// ---- POUs/BaseModule/ActionModule/motorModule/visu/motionModuleP1.TcVIS
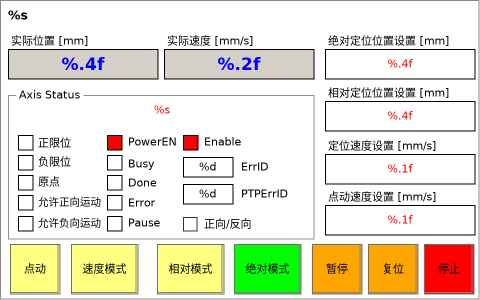
VISUALIZATION motionModuleP1  // 480x300
VAR_IN_OUT
	userData: motionModuleDataHMI;	
END_VAR
    Button (10,244 50x50), "点动", input disabled if: NOT userData.jogCondition OR NOT userData.ctrlModeCondition
        tap userData.manJogGo
    Button (157,244 67x50), "相对模式", tooltip "Please keep pressing to trigger", input disabled if: NOT userData.relCondition OR NOT userData.ctrlModeCondition
        tap userData.manRelGo
    Button (234,244 67x50), "绝对模式", tooltip "Please keep pressing to trigger", input disabled if: NOT userData.absCondition OR NOT userData.ctrlModeCondition
        tap userData.manABSGo
    Button (424,244 50x50), "停止"
        tap userData.stop
    Rectangle (8,49 150x30), "%.4f", text variable: userData.actualPos
    Rectangle (8,26 150x30), "实际位置 [mm]"
    Rectangle (164,49 150x30), "%.2f", text variable: userData.actualVel
    Rectangle (164,26 150x30), "实际速度 [mm/s]"
    Rectangle (325,79 145x28), "相对定位位置设置 [mm]"
    Rectangle (325,26 150x30), "绝对定位位置设置 [mm]"
    Rectangle (325,131 150x30), "定位速度设置 [mm/s]"
    GroupBox (8,87 306x152), "Axis Status"
        Rectangle (99,48 15x15), colour toggle: userData.powerEnable
        Rectangle (117,44 64x22), "PowerEN"
        Rectangle (10,48 15x15), colour toggle: userData.forwardLimitSwitch
        Rectangle (10,68 15x15), colour toggle: userData.backwardsLimitSwitch
        Rectangle (10,88 15x15), colour toggle: userData.dogPointSwitch
        Rectangle (27,84 64x22), "原点"
        Rectangle (99,68 15x15), colour toggle: userData.busy
        Rectangle (117,66 64x22), "Busy"
        Rectangle (230,69 46x22), "ErrID"
        Rectangle (27,104 67x22), "允许正向运动"
        Rectangle (10,108 15x15), colour toggle: userData.forwardEnable
        Rectangle (27,125 67x22), "允许负向运动"
        Rectangle (10,129 15x15), colour toggle: userData.backwardsEnable
        Rectangle (117,85 64x22), "Done"
        Rectangle (117,105 64x22), "Error"
        Rectangle (175,97 50x20), "%d", text variable: userData.PTPErrID
        Rectangle (99,129 15x15), colour toggle: userData.oPause
        Rectangle (117,125 64x22), "Pause"
        Rectangle (27,45 68x22), "正限位"
        Rectangle (27,64 64x22), "负限位"
        Rectangle (175,70 50x20), "%d", text variable: userData.errID
        Rectangle (175,48 15x15), colour toggle: userData.enable
        Rectangle (230,96 64x22), "PTPErrID"
        Rectangle (99,88 15x15), colour toggle: userData.done
        Rectangle (99,108 15x15), colour toggle: userData.error
        Checkbox (173,122 130x30), "正向/反向", variable: userData.choiceOfDirection
        Rectangle (193,44 52x22), "Enable"
    Rectangle (12,100 300x20), "%s", text variable: userData.errTxt
    Rectangle (325,49 150x30), "%.4f", text variable: userData.manABSPos, input disabled if: Not userData.goHomeDone
        OnMouseDown: write the text variable via Edit
    Rectangle (325,101 150x30), "%.4f", text variable: userData.manRelDis
        OnMouseDown: write the text variable via Edit
    Rectangle (325,154 150x30), "%.1f", text variable: userData.manVel
        OnMouseDown: write the text variable via Edit
    Rectangle (325,182 150x30), "点动速度设置 [mm/s]"
    Rectangle (325,205 150x30), "%.1f", text variable: userData.manJogVel
        OnMouseDown: write the text variable via Edit
    Button (71,244 67x50), "速度模式", invisible if: FALSE, input disabled if: NOT userData.velCondition OR NOT userData.ctrlModeCondition
        tap userData.manVelGo
    Button (368,244 50x50), "复位"
        tap userData.reset
    Rectangle (5,5 467x20), "%s", text variable: userData.nameTXT
    Button (312,244 50x50), "暂停", colour toggle: userData.oPause, input disabled if: NOT userData.ctrlModeCondition
        tap userData.pauseB
END_VISUALIZATION

// ---- POUs/BaseModule/ActionModule/motorModule/visu/motionModuleP2.TcVIS
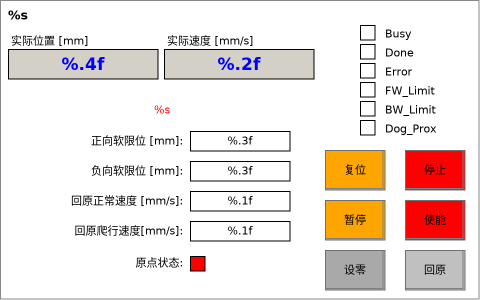
VISUALIZATION motionModuleP2  // 480x300
VAR_IN_OUT
	userData: motionModuleDataHMI;
END_VAR
    Rectangle (36,126 150x30), "正向软限位 [mm]:"
    Rectangle (190,131 100x20), "%.3f", text variable: userData.softPLimitPos, input disabled if: TRUE
        OnMouseDown: write the text variable via Edit
    Rectangle (36,156 150x30), "负向软限位 [mm]:"
    Rectangle (190,161 100x20), "%.3f", text variable: userData.softNLimitPos, input disabled if: TRUE
        OnMouseDown: write the text variable via Edit
    Rectangle (190,191 100x20), "%.1f", text variable: userData.goHomeVel
        OnMouseDown: write the text variable via Edit
    Button (405,250 60x40), "回原", colour toggle: userData.goHomeDone, input disabled if: NOT userData.homeCondition OR NOT userData.ctrlModeCondition
        tap userData.goHomeGo
    Rectangle (190,221 100x20), "%.1f", text variable: userData.goHomeVelSlow
        OnMouseDown: write the text variable via Edit
    Rectangle (36,186 150x30), "回原正常速度 [mm/s]:"
    Rectangle (27,216 159x30), "回原爬行速度[mm/s]:"
    Rectangle (79,248 107x30), "原点状态:"
    Rectangle (8,49 150x30), "%.4f", text variable: userData.actualPos
    Rectangle (8,26 150x30), "实际位置 [mm]"
    Rectangle (164,49 150x30), "%.2f", text variable: userData.actualVel
    Rectangle (164,26 150x30), "实际速度 [mm/s]"
    Rectangle (360,82 15x15), colour toggle: userData.forwardLimitSwitch
    Rectangle (360,101 15x15), colour toggle: userData.backwardsLimitSwitch
    Rectangle (360,120 15x15), colour toggle: userData.dogPointSwitch
    Rectangle (382,80 64x22), "FW_Limit"
    Rectangle (382,99 64x22), "BW_Limit"
    Rectangle (382,118 64x22), "Dog_Prox"
    Button (405,200 60x40), "使能", colour toggle: userData.powerEnable, input disabled if: NOT userData.ctrlModeCondition
        tap userData.power
    Button (325,250 60x40), "设零", invisible if: TRUE, input disabled if: NOT userData.setCondition OR NOT userData.ctrlModeCondition
        tap userData.setZero
    Button (325,200 60x40), "暂停", colour toggle: userData.oPause, input disabled if: NOT userData.ctrlModeCondition
        tap userData.pauseB
    Rectangle (190,256 15x15), colour toggle: userData.goHomeDone
    Rectangle (12,100 300x20), "%s", text variable: userData.errTxt
    Rectangle (5,5 467x20), "%s", text variable: userData.nameTXT
    Button (405,150 60x40), "停止"
        tap userData.stop
    Button (325,150 60x40), "复位"
        tap userData.reset
    Rectangle (360,25 15x15), colour toggle: userData.busy
    Rectangle (382,23 64x22), "Busy"
    Rectangle (382,42 64x22), "Done"
    Rectangle (382,61 64x22), "Error"
    Rectangle (360,44 15x15), colour toggle: userData.done
    Rectangle (360,63 15x15), colour toggle: userData.error
END_VISUALIZATION

// ---- POUs/BaseModule/ActionModule/motorModule/visu/motionModuleP3.TcVIS
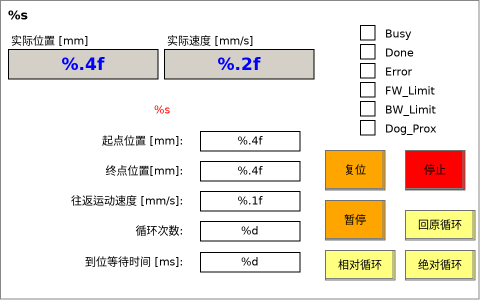
VISUALIZATION motionModuleP3  // 480x300
VAR_IN_OUT
	userData: motionModuleDataHMI;	
END_VAR
    Rectangle (36,126 150x30), "起点位置 [mm]:"
    Rectangle (36,156 150x30), "终点位置[mm]:"
    Rectangle (36,186 150x30), "往返运动速度 [mm/s]:"
    Rectangle (27,216 159x30), "循环次数:"
    Rectangle (8,49 150x30), "%.4f", text variable: userData.actualPos
    Rectangle (8,26 150x30), "实际位置 [mm]"
    Rectangle (164,49 150x30), "%.2f", text variable: userData.actualVel
    Rectangle (164,26 150x30), "实际速度 [mm/s]"
    Rectangle (12,100 300x20), "%s", text variable: userData.errTxt
    Rectangle (5,5 467x20), "%s", text variable: userData.nameTXT
    Rectangle (200,131 100x20), "%.4f", text variable: userData.loopFirstPoint
        OnMouseDown: write the text variable via Edit
    Rectangle (200,161 100x20), "%.4f", text variable: userData.loopSecondPoint
        OnMouseDown: write the text variable via Edit
    Rectangle (200,191 100x20), "%.1f", text variable: userData.loopGoVel
        OnMouseDown: write the text variable via Edit, min 0
    Rectangle (200,221 100x20), "%d", text variable: userData.loopCycle
        OnMouseDown: write the text variable via Edit, min 0
    Button (325,250 70x30), "相对循环", tooltip "Please keep pressing to trigger the relative motion loop", input disabled if: NOT userData.loopRelCondition OR NOT userData.ctrlModeCondition
        tap userData.loopRelGo
    Button (405,250 70x30), "绝对循环", tooltip "Please keep pressing to trigger the absolute motion loop", input disabled if: NOT userData.loopAbsCondition OR NOT userData.ctrlModeCondition
        tap userData.loopAbsGo
    Rectangle (27,247 159x30), "到位等待时间 [ms]:"
    Rectangle (200,252 100x20), "%d", text variable: userData.loopWatingTime
        OnMouseDown: write the text variable via Edit, min 0
    Button (405,150 60x40), "停止"
        tap userData.stop
    Button (325,150 60x40), "复位"
        tap userData.reset
    Rectangle (360,82 15x15), colour toggle: userData.forwardLimitSwitch
    Rectangle (360,101 15x15), colour toggle: userData.backwardsLimitSwitch
    Rectangle (360,120 15x15), colour toggle: userData.dogPointSwitch
    Rectangle (382,80 64x22), "FW_Limit"
    Rectangle (382,99 64x22), "BW_Limit"
    Rectangle (382,118 64x22), "Dog_Prox"
    Rectangle (360,25 15x15), colour toggle: userData.busy
    Rectangle (382,23 64x22), "Busy"
    Rectangle (382,42 64x22), "Done"
    Rectangle (382,61 64x22), "Error"
    Rectangle (360,44 15x15), colour toggle: userData.done
    Rectangle (360,63 15x15), colour toggle: userData.error
    Button (325,200 60x40), "暂停", colour toggle: userData.oPause, input disabled if: NOT userData.ctrlModeCondition
        tap userData.pauseB
    Button (405,210 70x30), "回原循环", tooltip "Please keep pressing to trigger the absolute motion loop", input disabled if: NOT userData.loopHomeToAbsCondition OR NOT userData.ctrlModeCondition
        tap userData.loopHomeToPosGo
END_VISUALIZATION

// ---- POUs/BaseModule/ActionModule/TMPModule/visu/TMPModuleVisu.TcVIS
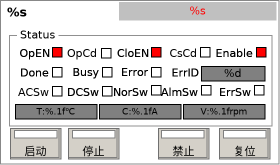
VISUALIZATION TMPModuleVisu  // 280x165
VAR_IN_OUT
	userData: TMPHMIStruts;
END_VAR
    Button (10,128 51x31), "启动", input disabled if: NOT userData.HMIEnable
        tap userData.open
    Rectangle (14,130 43x8), colour toggle: userData.openRelay
    GroupBox (9,27 263x99), "Status"
        RoundedRectangle (43,40 10x10), colour toggle: userData.done
        RoundedRectangle (247,20 10x10), colour toggle: userData.enable
        RoundedRectangle (93,40 10x10), colour toggle: userData.busy
        RoundedRectangle (142,40 10x10), colour toggle: userData.error
        Rectangle (192,39 64x15), "%d", text variable: userData.errID
        Label (7,20 37x13), "OpEN"
        RoundedRectangle (43,20 10x10), colour toggle: userData.enableOpen
        Label (106,20 37x13), "CloEN"
        RoundedRectangle (142,20 10x10), colour toggle: userData.enableClose
        Label (208,20 39x13), "Enable"
        Label (160,39 33x14), "ErrID"
        Label (112,39 30x13), "Error"
        Label (63,39 30x13), "Busy"
        Label (10,38 33x16), "Done"
        RoundedRectangle (43,59 10x10), colour toggle: userData.AccAprSw
        RoundedRectangle (93,59 10x10), colour toggle: userData.DccAprSw
        Label (56,59 37x13), "DCSw"
        Label (105,59 37x13), "NorSw"
        RoundedRectangle (142,58 10x10), colour toggle: userData.NormalAprSw
        Label (152,59 40x13), "AlmSw"
        RoundedRectangle (192,58 10x10), colour toggle: userData.AlmAprSw
        Label (208,59 37x13), "ErrSw"
        RoundedRectangle (245,58 10x10), colour toggle: userData.ErrorAprSw
        Rectangle (6,77 82x15), "T:%.1f℃", text variable: userData.temperature, input disabled if: true
        Rectangle (90,77 82x15), "C:%.1fA", text variable: userData.current, input disabled if: true
        Rectangle (174,77 82x15), "V:%.1frpm", text variable: userData.speed, input disabled if: true
        Label (157,20 34x13), "CsCd"
    RoundedRectangle (52,67 10x10), colour toggle: userData.done
    RoundedRectangle (256,47 10x10), colour toggle: userData.enable
    RoundedRectangle (102,67 10x10), colour toggle: userData.busy
    RoundedRectangle (151,67 10x10), colour toggle: userData.error
    Rectangle (201,66 64x15), "%d", text variable: userData.errID, input disabled if: true
    Label (16,47 37x13), "OpEN"
    RoundedRectangle (52,47 10x10), colour toggle: userData.enableOpen
    Label (115,47 37x13), "CloEN"
    RoundedRectangle (151,47 10x10), colour toggle: userData.enableClose
    Label (217,47 39x13), "Enable"
    Label (169,66 33x14), "ErrID"
    Label (121,66 30x13), "Error"
    Label (72,66 30x13), "Busy"
    Label (19,65 33x16), "Done"
    RoundedRectangle (52,86 10x10), colour toggle: userData.AccAprSw
    RoundedRectangle (102,86 10x10), colour toggle: userData.DccAprSw
    Label (65,86 37x13), "DCSw"
    Label (114,86 37x13), "NorSw"
    RoundedRectangle (151,85 10x10), colour toggle: userData.NormalAprSw
    Label (161,86 40x13), "AlmSw"
    RoundedRectangle (201,85 10x10), colour toggle: userData.AlmAprSw
    Label (217,86 37x13), "ErrSw"
    RoundedRectangle (254,85 10x10), colour toggle: userData.ErrorAprSw
    Button (219,128 51x31), "复位"
        tap userData.reset
    Rectangle (223,130 43x8), colour toggle: userData.resetRelay
    Rectangle (4,2 114x20), "%s", text variable: userData.nameTXT
    Button (68,128 51x31), "停止"
        tap userData.close
    Rectangle (72,130 43x8), colour toggle: userData.closeRelay
    Label (15,86 37x13), "ACSw"
    Button (158,128 51x31), "禁止"
        tap userData.stop
    Rectangle (161,130 43x8)
    Rectangle (119,2 157x18), "%s", text variable: userData.errTXT
    Label (64,47 36x13), "OpCd"
    RoundedRectangle (101,48 10x10), colour toggle: userData.opencondition
    RoundedRectangle (200,47 10x10), colour toggle: userData.closecondition
END_VISUALIZATION

// ---- POUs/BaseModule/ActionModule/VPEModule/visu/VPEModuleVis.TcVIS
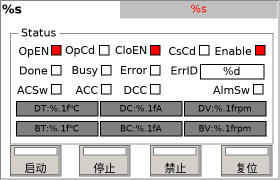
VISUALIZATION VPEModuleVis  // 280x180
VAR_IN_OUT
	userData: VPEHMIStruts;
END_VAR
    Button (10,145 51x31), "启动", input disabled if: NOT userData.HMIEnable
        tap userData.open
    Rectangle (14,147 43x8), colour toggle: userData.openRelay
    GroupBox (10,25 263x119), "Status"
        RoundedRectangle (41,40 10x10), colour toggle: userData.done
        RoundedRectangle (245,20 10x10), colour toggle: userData.enable
        RoundedRectangle (91,40 10x10), colour toggle: userData.busy
        RoundedRectangle (140,40 10x10), colour toggle: userData.error
        Rectangle (190,39 64x15), "%d", text variable: userData.errID
        Label (5,20 37x13), "OpEN"
        RoundedRectangle (41,20 10x10), colour toggle: userData.enableOpen
        RoundedRectangle (140,20 10x10), colour toggle: userData.enableClose
        Label (206,20 39x13), "Enable"
        Label (158,39 33x14), "ErrID"
        Label (110,39 30x13), "Error"
        Label (61,39 30x13), "Busy"
        Label (8,38 33x16), "Done"
        RoundedRectangle (41,59 10x10), colour toggle: userData.AccAprSw
        Label (203,59 40x13), "AlmSw"
        RoundedRectangle (243,59 10x10), colour toggle: userData.AlmAprSw
        Rectangle (6,96 82x15), "BT:%.1f℃", text variable: userData.BoosterTemperature, input disabled if: true
        RoundedRectangle (140,59 10x10), colour toggle: userData.Dccing
        RoundedRectangle (91,59 10x10), colour toggle: userData.Accing
        Label (52,19 36x13), "OpCd"
        RoundedRectangle (89,20 10x10), colour toggle: userData.opencondition
        Label (103,19 37x13), "CloEN"
    Button (221,145 51x31), "复位"
        tap userData.reset
    Rectangle (225,147 43x8), colour toggle: userData.reset
    Rectangle (-1,-1 119x20), "%s", text variable: userData.nameTXT
    Button (79,145 51x31), "停止"
        tap userData.close
    Rectangle (83,147 43x8)
    Label (14,84 37x13), "ACSw"
    Button (150,145 51x31), "禁止"
        tap userData.stop
    Rectangle (16,101 82x15), "DT:%.1f℃", text variable: userData.DryPumpTemperature, input disabled if: true
    Rectangle (100,101 82x15), "DC:%.1fA", text variable: userData.DryPumpCurrent, input disabled if: true
    Rectangle (184,101 82x15), "DV:%.1frpm", text variable: userData.DryPumpSpeed, input disabled if: true
    Rectangle (153,147 43x8)
    Rectangle (100,121 82x15), "BC:%.1fA", text variable: userData.BoosterCurrent, input disabled if: true
    Rectangle (184,121 82x15), "BV:%.1frpm", text variable: userData.BoosterSpeed, input disabled if: true
    Rectangle (120,0 157x18), "%s", text variable: userData.errTXT
    Label (113,84 37x13), "DCC"
    Label (70,84 31x13), "ACC"
    RoundedRectangle (199,45 10x10), colour toggle: userData.closecondition
    Label (165,45 34x13), "CsCd"
END_VISUALIZATION

// ---- POUs/BaseModule/IO/visu/IOBase_Show_New.TcVIS
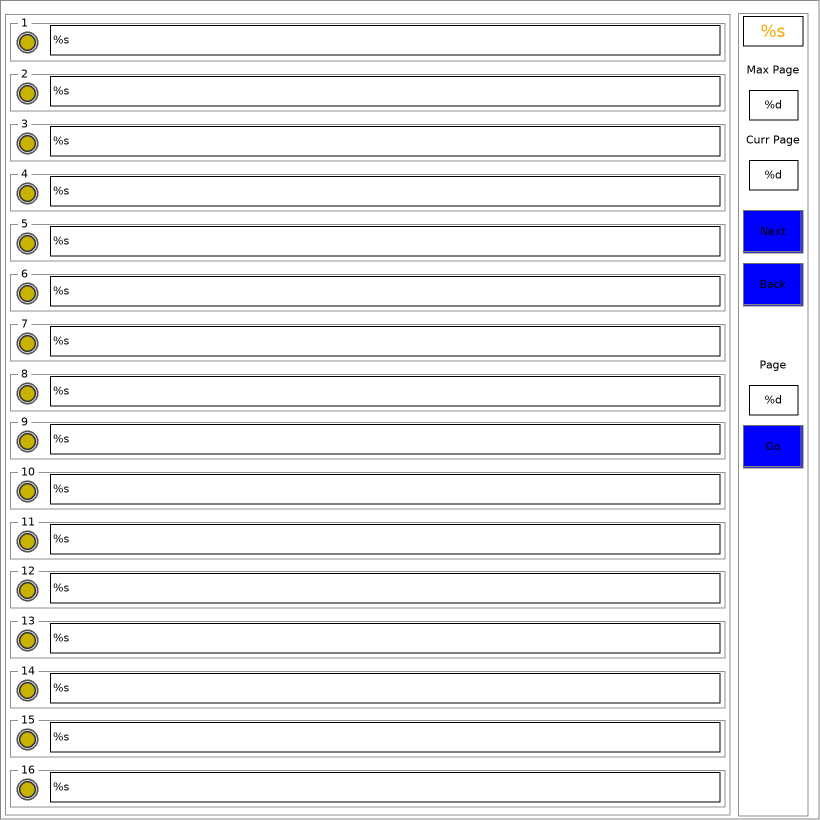
VISUALIZATION IOBase_Show_New  // 820x820
VAR_IN_OUT
	userData:ST_IOBase_Show_HMI;
END_VAR
    GroupBox (5,6 725x809)
        GroupBox (5,9 715x46), "1"
            Lamp1 (5,15 25x25), variable: userData.bIO[1], style: Lamp-Lamp1-Yellow
            Rectangle (40,10 670x30), "%s", text variable: userData.sInfor[1]
        GroupBox (5,60 715x45), "2"
            Lamp1 (5,15 25x25), variable: userData.bIO[2], style: Lamp-Lamp1-Yellow
            Rectangle (40,10 670x30), "%s", text variable: userData.sInfor[2]
        GroupBox (5,110 715x45), "3"
            Lamp1 (5,15 25x25), variable: userData.bIO[3], style: Lamp-Lamp1-Yellow
            Rectangle (40,10 670x30), "%s", text variable: userData.sInfor[3]
        GroupBox (5,160 715x45), "4"
            Lamp1 (5,15 25x25), variable: userData.bIO[4], style: Lamp-Lamp1-Yellow
            Rectangle (40,10 670x30), "%s", text variable: userData.sInfor[4]
        GroupBox (5,210 715x45), "5"
            Lamp1 (5,15 25x25), variable: userData.bIO[5], style: Lamp-Lamp1-Yellow
            Rectangle (40,10 670x30), "%s", text variable: userData.sInfor[5]
        GroupBox (5,260 715x45), "6"
            Lamp1 (5,15 25x25), variable: userData.bIO[6], style: Lamp-Lamp1-Yellow
            Rectangle (40,10 670x30), "%s", text variable: userData.sInfor[6]
        GroupBox (5,310 715x45), "7"
            Lamp1 (5,15 25x25), variable: userData.bIO[7], style: Lamp-Lamp1-Yellow
            Rectangle (40,10 670x30), "%s", text variable: userData.sInfor[7]
        GroupBox (5,360 715x45), "8"
            Lamp1 (5,15 25x25), variable: userData.bIO[8], style: Lamp-Lamp1-Yellow
            Rectangle (40,10 670x30), "%s", text variable: userData.sInfor[8]
        GroupBox (5,408 715x45), "9"
            Lamp1 (5,15 25x25), variable: userData.bIO[9], style: Lamp-Lamp1-Yellow
            Rectangle (40,10 670x30), "%s", text variable: userData.sInfor[9]
        GroupBox (5,458 715x45), "10"
            Lamp1 (5,15 25x25), variable: userData.bIO[10], style: Lamp-Lamp1-Yellow
            Rectangle (40,10 670x30), "%s", text variable: userData.sInfor[10]
        GroupBox (5,508 715x45), "11"
            Lamp1 (5,15 25x25), variable: userData.bIO[11], style: Lamp-Lamp1-Yellow
            Rectangle (40,10 670x30), "%s", text variable: userData.sInfor[11]
        GroupBox (5,557 715x45), "12"
            Lamp1 (5,15 25x25), variable: userData.bIO[12], style: Lamp-Lamp1-Yellow
            Rectangle (40,10 670x30), "%s", text variable: userData.sInfor[12]
        GroupBox (5,607 715x45), "13"
            Lamp1 (5,15 25x25), variable: userData.bIO[13], style: Lamp-Lamp1-Yellow
            Rectangle (40,10 670x30), "%s", text variable: userData.sInfor[13]
        GroupBox (5,657 715x45), "14"
            Lamp1 (5,15 25x25), variable: userData.bIO[14], style: Lamp-Lamp1-Yellow
            Rectangle (40,10 670x30), "%s", text variable: userData.sInfor[14]
        GroupBox (5,706 715x45), "15"
            Lamp1 (5,15 25x25), variable: userData.bIO[15], style: Lamp-Lamp1-Yellow
            Rectangle (40,10 670x30), "%s", text variable: userData.sInfor[15]
        GroupBox (5,756 715x45), "16"
            Lamp1 (5,15 25x25), variable: userData.bIO[16], style: Lamp-Lamp1-Yellow
            Rectangle (40,10 670x30), "%s", text variable: userData.sInfor[16]
    GroupBox (738,5 70x811)
        Button (5,205 60x43), "Next"
            tap userData.bNextPage
        Button (5,258 60x43), "Back"
            tap userData.bBackPage
        Rectangle (11,85 49x30), "%d", text variable: userData.iMaxPage
        Rectangle (11,155 49x30), "%d", text variable: userData.iCurrPage
        Rectangle (11,380 49x30), "%d", text variable: userData.iTargerPage
            OnMouseUp: write the text variable via Default, min 1, max 99
        Button (5,420 60x43), "Go"
            tap userData.bTargerPage
        Label (5,50 60x30), "Max Page"
        Label (5,120 60x30), "Curr Page"
        Label (5,345 60x30), "Page"
        Rectangle (5,11 60x30), "%s", text variable: userData.sIOType
END_VISUALIZATION

// ---- POUs/BaseModule/MainFrame/MainFrame.TcVIS
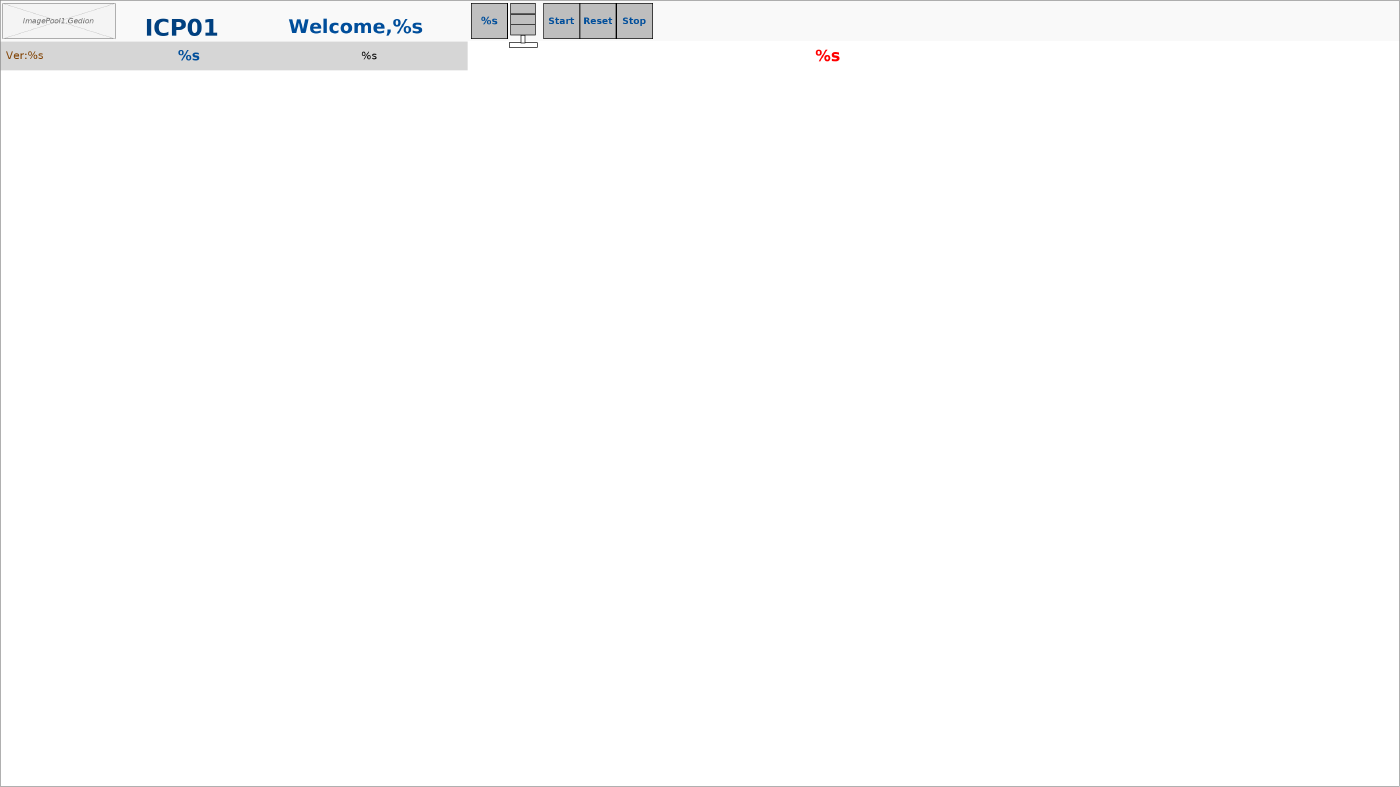
VISUALIZATION MainFrame  // 1920x1080, background image ImagePool1.background
VAR_IN_OUT
	userData:MainFram;
END_VAR
    Rectangle (0,57 641x39)
    Rectangle (373,57 267x39), "%s", text variable: userData.ShowTime
    Rectangle (646,57 979x39), "%s", text variable: userData.ErrWTxtShow, invisible if: Not (gRunningState=RunningStatus.eErrorState)
    Rectangle (5,57 142x38), "Ver:%s", text variable: userData.versions
    Rectangle (0,0 1920x56)
    InvisibleInput (0,0 1x12)
    InvisibleInput (0,0 1x1)
    Rectangle (363,20 250x33), "Welcome,%s", text variable: gCurrentUser
    Image (3,4 155x49), image: ImagePool1.Gedion
    Rectangle (173,23 175x30), "ICP01"
    Group (698,4 45x49)
        Rectangle (2,0 34x15), colour toggle: userData.RedLamp
        Rectangle (2,15 34x15), colour toggle: userData.YellowLamp
        Rectangle (2,29 34x15), colour toggle: userData.GreenLamp
        Rectangle (0,54 39x7)
        Rectangle (16,44 6x11)
    Rectangle (745,4 50x49), "Start", colour toggle: userData.StartLamp
        tap userData.Start
    Rectangle (795,4 50x49), "Reset", colour toggle: userData.ResetLamp
        tap userData.Reset
    Rectangle (845,4 50x49), "Stop", colour toggle: userData.StopLamp
        tap userData.Stop
    Rectangle (646,4 50x49), "%s", tooltip "A:Auto Running E:Error Running H:Homing M:Manual Running P:Pause Running S:Stop Running", text variable: userData.RunStateTxt
    Rectangle (153,57 213x39), "%s", text variable: fbMachineState.RunStateTxt
END_VISUALIZATION

// ---- POUs/BaseModule/PrintLogModule_EX/visu/showInfo_Auto.TcVIS
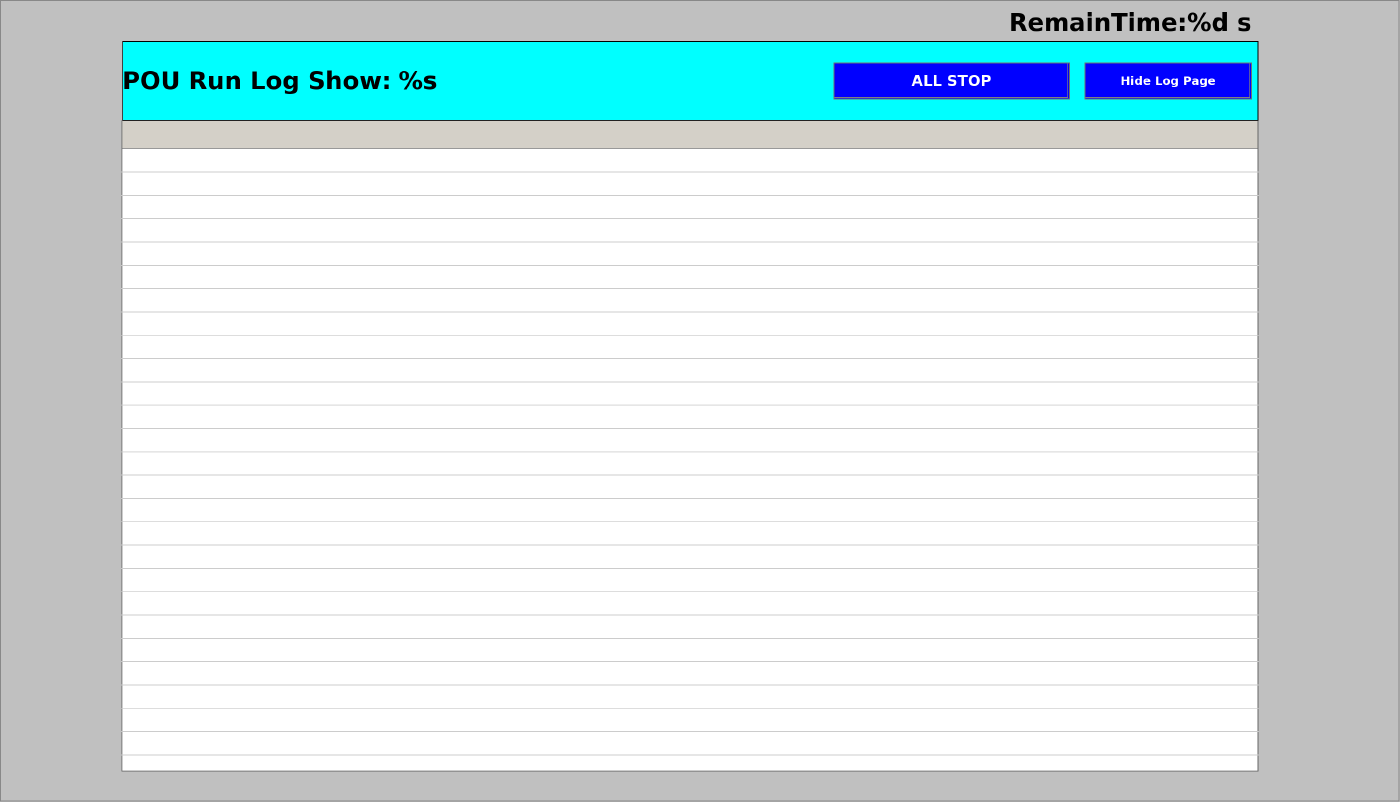
VISUALIZATION showInfo_Auto  // 1500x860
VAR_IN_OUT
	userData: printLogModule_EX_DataHMI;
END_VAR
    Rectangle (0,0 1500x860)
    Table (130,129 1218x698), data array: userData.logStrData
        p1128707560: cNumLength_showInof
        p3854506369: userData.logStrData[INDEX].sTime
        p1892666644: userData.logStrData[INDEX].msg
        p511219082: Information
    RoundedRectangle (131,44 1217x85)
    Label (133,57 285x59), "POU Run Log Show:"
    Button (1162,67 179x39), "Hide Log Page"
        OnMouseClick: execute { gShowPOURunLog:=NOT gShowPOURunLog; }
    Button (893,67 253x39), "ALL STOP"
        tap MainRunPOU.AllAbort
        OnMouseClick: execute {
            gShowPOURunLog:=NOT gShowPOURunLog;
            gCtrlMode:=ControlMode.eManualCtrMode;
            IF RunningStatus.eErrorState<>gRunningState THEN
            	gRunningState:=RunningStatus.eManualState;
            END_IF
        }
    Rectangle (424,51 443x71), "%s", text variable: gShowLogTextTitle
    Rectangle (1003,3 341x42), "RemainTime:%d s", text variable: gCO_ControlRFRMTime, invisible if: NOT S_CO_ControlRF.busy
END_VISUALIZATION

// ---- POUs/BaseModule/PrintLogModule_EX/visu/showInfo.TcVIS
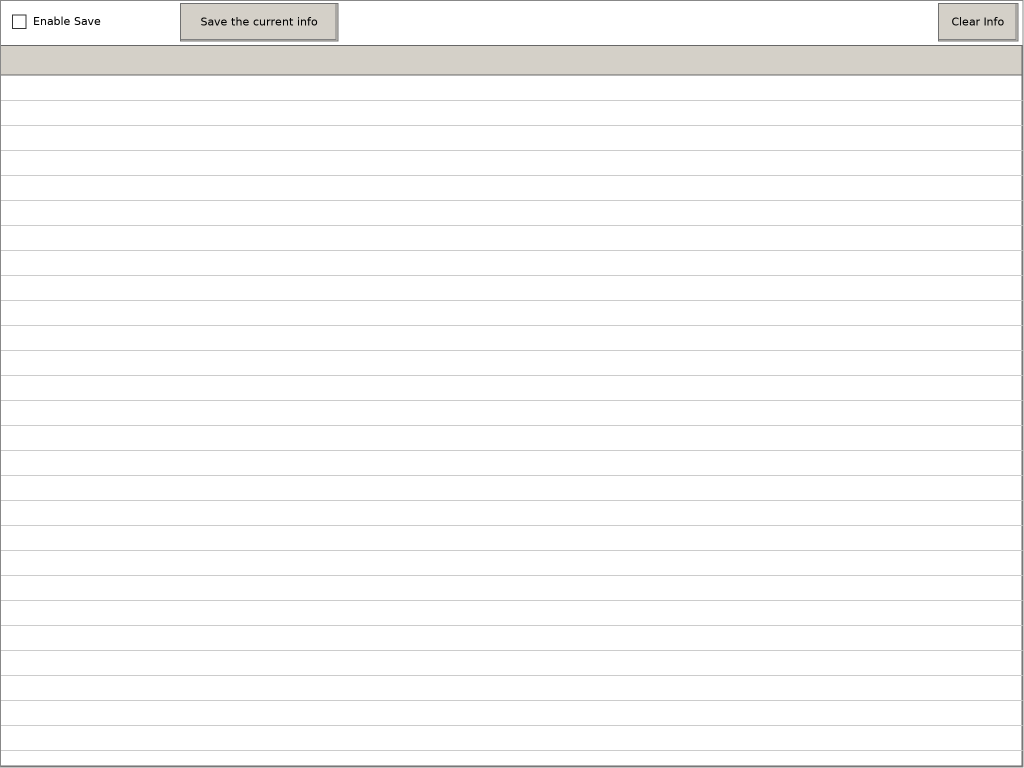
VISUALIZATION showInfo  // 1024x768
VAR_IN_OUT
	userData: printLogModule_EX_DataHMI;
END_VAR
    Checkbox (10,9 150x25), "Enable Save", variable: userData.enableSave
    Button (180,3 158x38), "Save the current info"
        tap userData.enableSaveShowLog
    Button (938,3 80x38), "Clear Info"
        tap userData.clearInformation
    Table (0,45 1022x721), data array: userData.logStrData
        p1128707560: cNumLength_showInof
        p3854506369: userData.logStrData[INDEX].sTime
        p1892666644: userData.logStrData[INDEX].msg
        p511219082: Information
END_VISUALIZATION

// ---- POUs/Other/HMI/Note.TcVIS
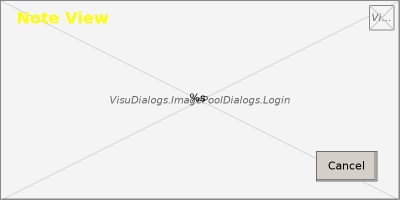
VISUALIZATION Note  // 400x200
VAR_IN_OUT
	noteHMI:NoteStruct;
END_VAR
    Image (0,0 400x200), image: VisuDialogs.ImagePoolDialogs.Login
    Rectangle (24,83 347x30), "%s", text variable: noteHMI.showText
    Button (316,151 61x30), "Cancel"
        OnMouseClick: execute { noteHMI.showFlag:=FALSE; }
    Image (369,5 25x25), image: VisuDialogs.ImagePoolDialogs.Delete
        OnMouseClick: execute { noteHMI.showFlag:=FALSE; }
    Label (5,3 116x30), "Note View"
END_VISUALIZATION

// ---- POUs/Other/HMI/WARM.TcVIS
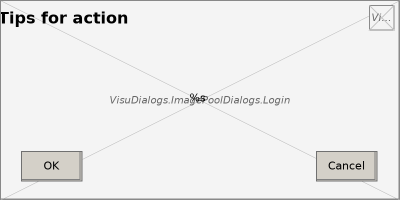
VISUALIZATION WARM  // 400x200
VAR_IN_OUT
	warmHMI:WARMStruct;
END_VAR
    Image (0,0 400x200), image: VisuDialogs.ImagePoolDialogs.Login
    Button (21,151 61x30), "OK"
        OnMouseClick: execute { warmHMI.bOK:=TRUE; warmHMI.showFlag:=FALSE; }
    Button (316,151 61x30), "Cancel"
        OnMouseClick: execute { warmHMI.bNO:=TRUE; warmHMI.showFlag:=FALSE; }
    Rectangle (24,83 347x30), "%s", text variable: warmHMI.showText
    Image (369,5 25x25), image: VisuDialogs.ImagePoolDialogs.Delete
        OnMouseClick: execute { warmHMI.bNO:=TRUE; warmHMI.showFlag:=FALSE; }
    Label (5,3 116x30), "Tips for action"
END_VISUALIZATION

// ---- VISUs/Editor/Manual.TcVIS
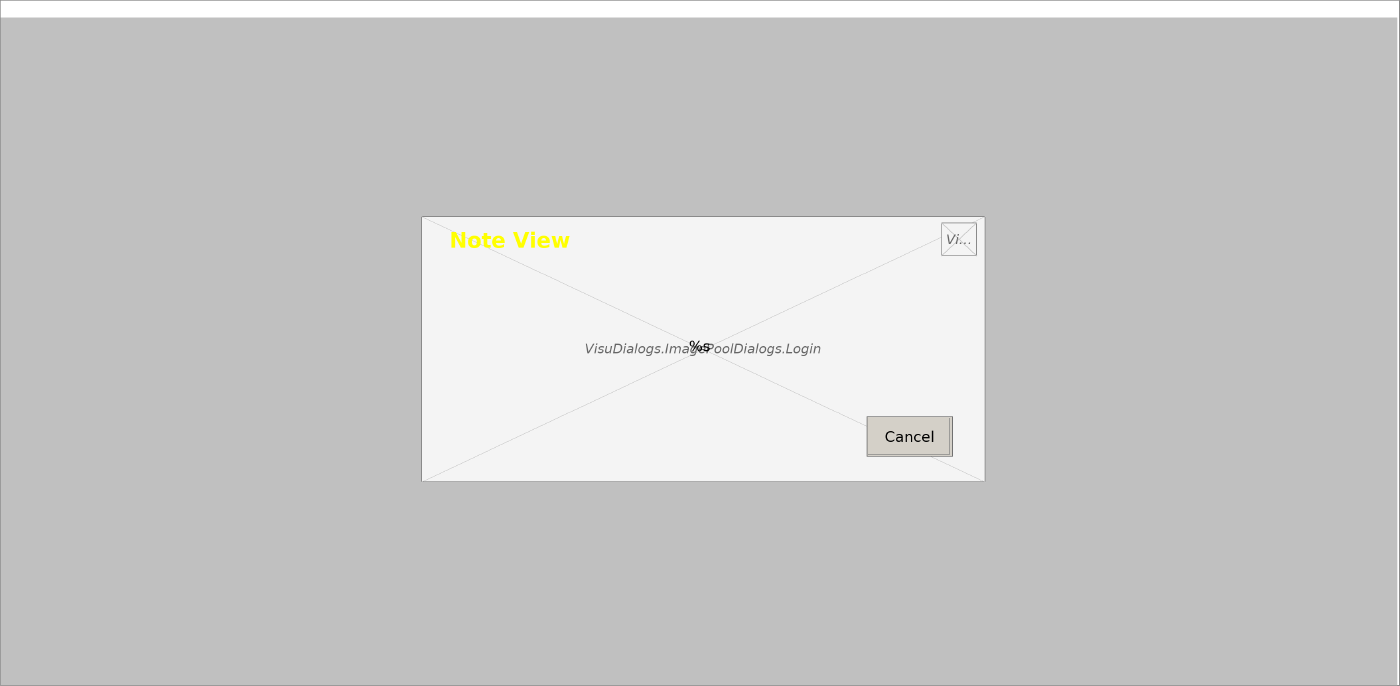
VISUALIZATION Manual  // 1755x860
    TabControl (0,0 1755x860), input disabled if: gWarmShowHMI.showFlag or gNoteShowHMI.showFlag or gPDVOpencondition or S_PDVSafeCtr.busy or gSPOUBusy
        shows Overview()
        shows Overview_Total()
        [0]: TabTitle=All Show
        [1]: TabTitle=Part Show
    Rectangle (0,22 1751x838), invisible if: (Not gWarmShowHMI.showFlag and Not gNoteShowHMI.showFlag) or gCtrlMode=ControlMode.eAutoCtrMode
    Frame (528,271 707x249), invisible if: NOT gWarmShowHMI.showFlag
        shows WARM(warmHMI := gWarmShowHMI)
    Frame (528,271 707x333), invisible if: Not gNoteShowHMI.showFlag or gCtrlMode=ControlMode.eAutoCtrMode
        shows Note(noteHMI := gNoteShowHMI)
END_VISUALIZATION

// ---- VISUs/Editor/Overview.TcVIS
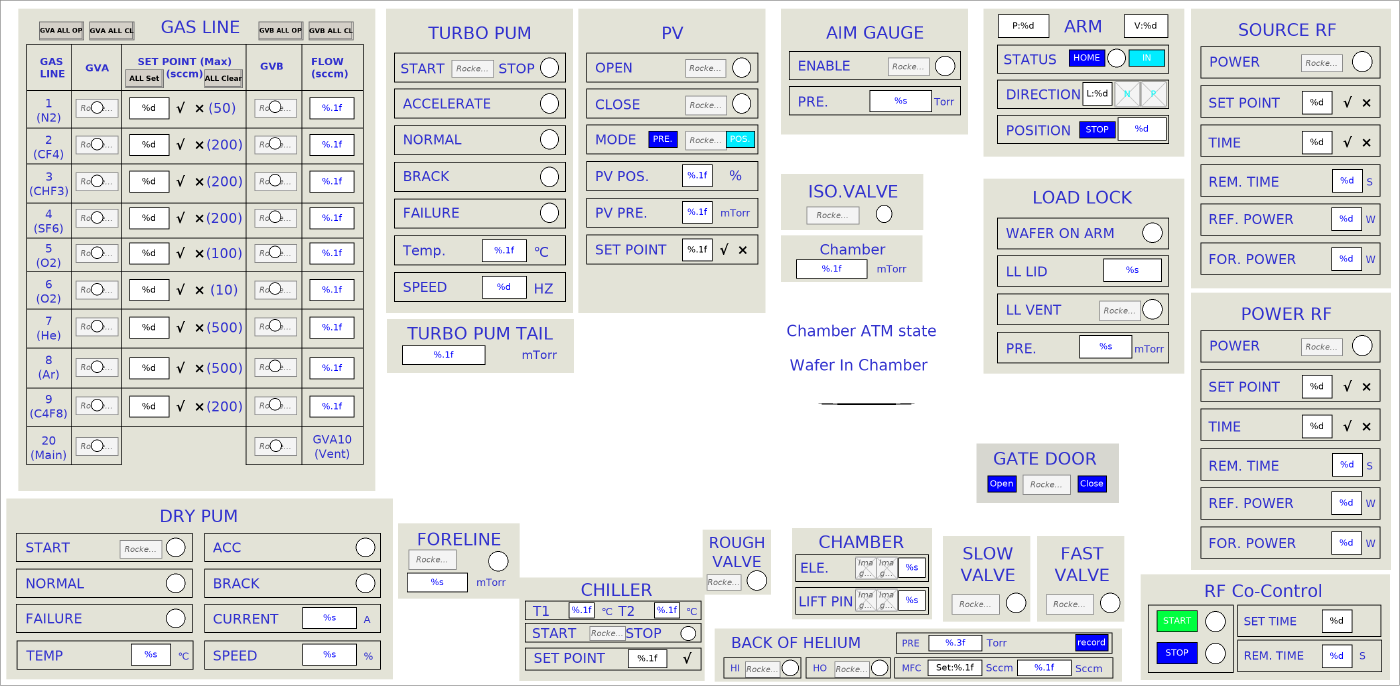
VISUALIZATION Overview  // 1755x860, background image ImagePool1.autoImg
    RoundedRectangle (23,11 447x604)
    RoundedRectangle (1233,11 251x185), colour toggle: NOT FuncModule_RS232_ARM.serialConnected, input disabled if: NOT FuncModule_RS232_ARM.serialConnected
    Label (1262,12 192x42), "ARM"
    RoundedRectangle (1250,56 215x36)
    RoundedRectangle (1250,100 215x36)
    Label (1258,108 110x21), "DIRECTION"
    RoundedRectangle (1250,144 215x36)
    Label (1258,153 96x21), "POSITION"
    RoundedRectangle (1340,62 45x21), "HOME", colour toggle: gICP.I_ARMHome, input disabled if: NOT FuncModule_RS232_ARM.serialConnected
        OnMouseClick: write the text variable via Default
        OnMouseClick: execute { gICP.ARM.Act_HOME(gICP.ARM.NoteHMI); }
    Label (1255,64 82x21), "STATUS"
    RoundedRectangle (1415,62 45x21), "IN", colour toggle: gICP.I_ARMHome or gICP.ARM.busy, input disabled if: NOT FuncModule_RS232_ARM.serialConnected
        OnMouseClick: write the text variable via Default
        OnMouseClick: execute { gICP.ARM.Act_IN(gICP.ARM.NoteHMI); }
    Ellipse (1388,61 23x23), colour toggle: gICP.ARM.busy or gICP.ARM.jogBusy
    Image (1397,102 32x32), "N", input disabled if: NOT FuncModule_RS232_ARM.serialConnected, image: VisuSymbols.Symbols.ArrowBoldLeft
        OnMouseClick: write the text variable via Default
        OnMouseClick: execute { gICP.ARM.Act_DirectionJog(_noteHMI:=gICP.ARM.NoteHMI,FALSE,gICp.ARM.setvel,gICP.ARM.jogsetlen); }
    Image (1430,102 32x32), "P", input disabled if: NOT FuncModule_RS232_ARM.serialConnected, image: VisuSymbols.Symbols.ArrowBoldRight
        OnMouseClick: write the text variable via Default
        OnMouseClick: execute { gICP.ARM.Act_DirectionJog(_noteHMI:=gICP.ARM.NoteHMI,TRUE,gICp.ARM.setvel,gICP.ARM.jogsetlen); }
    Group (993,662 175x114)
        RoundedRectangle (0,0 175x114)
        Label (19,2 136x31), "CHAMBER"
        RoundedRectangle (4,33 167x34)
        Label (7,40 59x20), "ELE."
        RoundedRectangle (4,74 167x34)
        Label (5,82 79x20), "LIFT PIN"
        Image (79,36 27x28), colour toggle: gICP.ElectrodeCyl.extend, image: ImagePool1.up
            OnMouseClick: write the text variable via Default
            OnMouseClick: execute { gICP.ElectrodeCyl.HMIItf.extend:=true; }
        Image (105,36 27x28), colour toggle: gICP.ElectrodeCyl.retract, image: ImagePool1.down
            OnMouseClick: write the text variable via Default
            OnMouseClick: execute { gICP.ElectrodeCyl.HMIItf.retract:=true; }
        Image (79,76 27x28), colour toggle: gICP.LiftPinCyl.extend, image: ImagePool1.up
            OnMouseClick: write the text variable via Default
            OnMouseClick: execute { gICP.LiftPinCyl.HMIItf.extend:=true; }
        Image (105,76 27x28), colour toggle: gICP.LiftPinCyl.retract, image: ImagePool1.down
            OnMouseClick: write the text variable via Default
            OnMouseClick: execute { gICP.LiftPinCyl.HMIItf.retract:=true; }
        RoundedRectangle (133,37 34x25), "%s", text variable: gICP.ElectrodeCyl.HMIItf.sensorShow
        RoundedRectangle (133,78 34x25), "%s", text variable: gICP.LiftPinCyl.HMIItf.sensorShow
    Line (33,55) (455,55)
    Line (33,582) (152,582)
    Line (33,113) (455,113)
    Line (33,160) (455,160)
    Line (33,205) (455,205)
    Line (33,254) (455,254)
    Line (33,298) (455,298)
    Line (33,340) (455,340)
    Line (33,387) (455,387)
    Line (33,486) (455,486)
    Line (33,55) (33,582)
    Line (89,55) (89,582)
    Line (152,55) (152,582)
    Line (308,55) (308,582)
    Line (378,55) (378,582)
    Line (455,55) (455,582)
    Label (40,13 423x42), "GAS LINE"
    Label (47,61 45x48), "GAS LINE"
    Label (104,61 42x48), "GVA"
    Label (387,61 59x48), "FLOW (sccm)"
    Label (323,59 45x48), "GVB"
    Label (168,61 127x48), "SET POINT (Max) (sccm)"
    RockerSwitch (95,124 53x23), variable: gICP.GVA1Valve.HMIItf.singleControl, behaviour: TOGGLE, style: Switch-RockerSwitch-Blue
    RockerSwitch (95,170 53x23), variable: gICP.GVA2Valve.HMIItf.singleControl, behaviour: TOGGLE, style: Switch-RockerSwitch-Blue
    RockerSwitch (95,216 53x23), variable: gICP.GVA3Valve.HMIItf.singleControl, behaviour: TOGGLE, style: Switch-RockerSwitch-Blue
    RockerSwitch (95,262 53x23), variable: gICP.GVA4Valve.HMIItf.singleControl, behaviour: TOGGLE, style: Switch-RockerSwitch-Blue
    RockerSwitch (95,306 53x23), variable: gICP.GVA5Valve.HMIItf.singleControl, behaviour: TOGGLE, style: Switch-RockerSwitch-Blue
    RockerSwitch (95,352 53x23), variable: gICP.GVA6Valve.HMIItf.singleControl, behaviour: TOGGLE, style: Switch-RockerSwitch-Blue
    RockerSwitch (95,449 53x23), variable: gICP.GVA8Valve.HMIItf.singleControl, behaviour: TOGGLE, style: Switch-RockerSwitch-Blue
    RockerSwitch (95,548 53x23), variable: gICP.GV20Valve_Main.HMIItf.singleControl, behaviour: TOGGLE, style: Switch-RockerSwitch-Blue
    RockerSwitch (319,124 53x23), variable: gICP.GVB1Valve.HMIItf.singleControl, behaviour: TOGGLE, style: Switch-RockerSwitch-Blue
    RockerSwitch (319,170 53x23), variable: gICP.GVB2Valve.HMIItf.singleControl, behaviour: TOGGLE, style: Switch-RockerSwitch-Blue
    RockerSwitch (319,216 53x23), variable: gICP.GVB3Valve.HMIItf.singleControl, behaviour: TOGGLE, style: Switch-RockerSwitch-Blue
    RockerSwitch (319,262 53x23), variable: gICP.GVB4Valve.HMIItf.singleControl, behaviour: TOGGLE, style: Switch-RockerSwitch-Blue
    RockerSwitch (319,306 53x23), variable: gICP.GVB5Valve.HMIItf.singleControl, behaviour: TOGGLE, style: Switch-RockerSwitch-Blue
    RockerSwitch (319,352 53x23), variable: gICP.GVB6Valve.HMIItf.singleControl, behaviour: TOGGLE, style: Switch-RockerSwitch-Blue
    RockerSwitch (319,449 53x23), variable: gICP.GVB8Valve.HMIItf.singleControl, behaviour: TOGGLE, style: Switch-RockerSwitch-Blue
    RoundedRectangle (388,448 56x27), "%.1f", text variable: gICP.MFC8.actflowFloat, colour toggle: NOT FuncModule_RS485_MFC.serialConnected
    RoundedRectangle (388,350 56x27), "%.1f", text variable: gICP.MFC6.actflowFloat, colour toggle: NOT FuncModule_RS485_MFC.serialConnected
    RoundedRectangle (388,304 56x27), "%.1f", text variable: gICP.MFC5.actflowFloat, colour toggle: NOT FuncModule_RS485_MFC.serialConnected
    RoundedRectangle (388,260 56x27), "%.1f", text variable: gICP.MFC4.actflowFloat, colour toggle: NOT FuncModule_RS485_MFC.serialConnected
    RoundedRectangle (388,214 56x27), "%.1f", text variable: gICP.MFC3.actflowFloat, colour toggle: NOT FuncModule_RS485_MFC.serialConnected
    RoundedRectangle (388,168 56x27), "%.1f", text variable: gICP.MFC2.actflowFloat, colour toggle: NOT FuncModule_RS485_MFC.serialConnected
    RoundedRectangle (388,122 56x27), "%.1f", text variable: gICP.MFC1.actflowFloat, colour toggle: NOT FuncModule_RS485_MFC.serialConnected
    Rectangle (162,122 50x27), "%d", text variable: gICP.MFC1.setFlow, colour toggle: gICP.MFC1.setdone
        OnMouseClick: write the text variable via Default
    Rectangle (215,122 23x27), "√", colour toggle: gICP.MFC1.setbusy
        OnMouseClick: write the text variable via Default
        OnMouseClick: execute { gICP.MFC1.MFCHMItif.set:=TRUE; }
    Rectangle (241,122 18x27), "×", colour toggle: gICP.MFC1.clearbusy
        OnMouseClick: write the text variable via Default
        OnMouseClick: execute { gICP.MFC1.MFCHMItif.clear:=TRUE; }
    Label (259,126 39x19), "(50)"
    Rectangle (162,168 50x27), "%d", text variable: gICP.MFC2.setFlow, colour toggle: gICP.MFC2.setdone
        OnMouseClick: write the text variable via Default
    Rectangle (215,168 23x27), "√", colour toggle: gICP.MFC2.setbusy
        OnMouseClick: write the text variable via Default
        OnMouseClick: execute { gICP.MFC2.MFCHMItif.set:=TRUE; }
    Rectangle (241,168 18x27), "×", colour toggle: gICP.MFC2.clearbusy
        OnMouseClick: write the text variable via Default
        OnMouseClick: execute { gICP.MFC2.MFCHMItif.clear:=TRUE; }
    Label (259,172 45x19), "(200)"
    Rectangle (162,214 50x27), "%d", text variable: gICP.MFC3.setFlow, colour toggle: gICP.MFC3.setdone
        OnMouseClick: write the text variable via Default
    Rectangle (215,214 23x27), "√", colour toggle: gICP.MFC3.setbusy
        OnMouseClick: write the text variable via Default
        OnMouseClick: execute { gICP.MFC3.MFCHMItif.set:=TRUE; }
    Rectangle (241,214 18x27), "×", colour toggle: gICP.MFC3.clearbusy
        OnMouseClick: write the text variable via Default
        OnMouseClick: execute { gICP.MFC3.MFCHMItif.clear:=TRUE; }
    Label (259,218 45x19), "(200)"
    Rectangle (162,260 50x27), "%d", text variable: gICP.MFC4.setFlow, colour toggle: gICP.MFC4.setdone
        OnMouseClick: write the text variable via Default
    Rectangle (215,260 23x27), "√", colour toggle: gICP.MFC4.setbusy
        OnMouseClick: write the text variable via Default
        OnMouseClick: execute { gICP.MFC4.MFCHMItif.set:=TRUE; }
    Rectangle (241,260 18x27), "×", colour toggle: gICP.MFC4.clearbusy
        OnMouseClick: write the text variable via Default
        OnMouseClick: execute { gICP.MFC4.MFCHMItif.clear:=TRUE; }
    Label (259,264 44x19), "(200)"
    Rectangle (162,304 50x27), "%d", text variable: gICP.MFC5.setFlow, colour toggle: gICP.MFC5.setdone
        OnMouseClick: write the text variable via Default
    Rectangle (215,304 23x27), "√", colour toggle: gICP.MFC5.setbusy
        OnMouseClick: write the text variable via Default
        OnMouseClick: execute { gICP.MFC5.MFCHMItif.set:=TRUE; }
    Rectangle (241,304 18x27), "×", colour toggle: gICP.MFC5.clearbusy
        OnMouseClick: write the text variable via Default
        OnMouseClick: execute { gICP.MFC5.MFCHMItif.clear:=TRUE; }
    Label (259,308 44x19), "(100)"
    Rectangle (162,350 50x27), "%d", text variable: gICP.MFC6.setFlow, colour toggle: gICP.MFC6.setdone
        OnMouseClick: write the text variable via Default
    Rectangle (215,350 23x27), "√", colour toggle: gICP.MFC6.setbusy
        OnMouseClick: write the text variable via Default
        OnMouseClick: execute { gICP.MFC6.MFCHMItif.set:=TRUE; }
    Rectangle (241,350 18x27), "×", colour toggle: gICP.MFC6.clearbusy
        OnMouseClick: write the text variable via Default
        OnMouseClick: execute { gICP.MFC6.MFCHMItif.clear:=TRUE; }
    Label (259,354 44x19), "(10)"
    Rectangle (162,448 50x27), "%d", text variable: gICP.MFC8.setFlow, colour toggle: gICP.MFC8.setdone
        OnMouseClick: write the text variable via Default
    Rectangle (215,448 23x27), "√", colour toggle: gICP.MFC8.setbusy
        OnMouseClick: write the text variable via Default
        OnMouseClick: execute { gICP.MFC8.MFCHMItif.set:=TRUE; }
    Rectangle (241,448 18x27), "×", colour toggle: gICP.MFC8.clearbusy
        OnMouseClick: write the text variable via Default
        OnMouseClick: execute { gICP.MFC8.MFCHMItif.clear:=TRUE; }
    Label (259,452 45x19), "(500)"
    Label (39,116 44x45), "1 (N2)"
    Label (39,162 44x45), "2 (CF4)"
    Label (39,255 44x45), "4 (SF6)"
    Label (35,208 53x45), "3 (CHF3)"
    Label (39,343 44x45), "6 (O2)"
    Label (39,298 44x45), "5 (O2)"
    Label (39,539 44x45), "20 (Main)"
    Label (39,438 44x45), "8 (Ar)"
    Ellipse (114,127 15x15), colour toggle: gICP.GVA1Valve.extRelay
    Ellipse (114,173 15x15), colour toggle: gICP.GVA2Valve.extRelay
    Ellipse (114,219 15x15), colour toggle: gICP.GVA3Valve.extRelay
    Ellipse (114,265 15x15), colour toggle: gICP.GVA4Valve.extRelay
    Ellipse (114,309 15x15), colour toggle: gICP.GVA5Valve.extRelay
    Ellipse (114,355 15x15), colour toggle: gICP.GVA6Valve.extRelay
    Ellipse (114,452 15x15), colour toggle: gICP.GVA8Valve.extRelay
    Ellipse (114,551 15x15), colour toggle: gICP.GV20Valve_Main.extRelay
    Ellipse (337,126 15x15), colour toggle: gICP.GVB1Valve.extRelay
    Ellipse (337,172 15x15), colour toggle: gICP.GVB2Valve.extRelay
    Ellipse (337,218 15x15), colour toggle: gICP.GVB3Valve.extRelay
    Ellipse (337,264 15x15), colour toggle: gICP.GVB4Valve.extRelay
    Ellipse (337,308 15x15), colour toggle: gICP.GVB5Valve.extRelay
    Ellipse (337,354 15x15), colour toggle: gICP.GVB6Valve.extRelay
    Ellipse (337,451 15x15), colour toggle: gICP.GVB8Valve.extRelay
    Line (33,534) (455,534)
    RockerSwitch (95,497 53x23), variable: gICP.GVA9Valve.HMIItf.singleControl, behaviour: TOGGLE, style: Switch-RockerSwitch-Blue
    RockerSwitch (319,497 53x23), variable: gICP.GVB9Valve.HMIItf.singleControl, behaviour: TOGGLE, style: Switch-RockerSwitch-Blue
    RoundedRectangle (388,496 56x27), "%.1f", text variable: gICP.MFC9.actflowFloat, colour toggle: NOT FuncModule_RS485_MFC.serialConnected
    Rectangle (162,496 50x27), "%d", text variable: gICP.MFC9.setFlow, colour toggle: gICP.MFC9.setdone
        OnMouseClick: write the text variable via Default
    Rectangle (215,496 23x27), "√", colour toggle: gICP.MFC9.setbusy
        OnMouseClick: write the text variable via Default
        OnMouseClick: execute { gICP.MFC9.MFCHMItif.set:=TRUE; }
    Rectangle (241,496 18x27), "×", colour toggle: gICP.MFC9.clearbusy
        OnMouseClick: write the text variable via Default
        OnMouseClick: execute { gICP.MFC9.MFCHMItif.clear:=TRUE; }
    Label (259,500 45x19), "(200)"
    Label (36,487 50x45), "9 (C4F8)"
    Ellipse (114,500 15x15), colour toggle: gICP.GVA9Valve.extRelay
    Ellipse (337,499 15x15), colour toggle: gICP.GVB9Valve.extRelay
    Line (33,436) (455,436)
    RockerSwitch (95,398 53x23), variable: gICP.GVA7Valve.HMIItf.singleControl, behaviour: TOGGLE, style: Switch-RockerSwitch-Blue
    RockerSwitch (319,398 53x23), variable: gICP.GVB7Valve.HMIItf.singleControl, behaviour: TOGGLE, style: Switch-RockerSwitch-Blue
    RoundedRectangle (388,397 56x27), "%.1f", text variable: gICP.MFC7.actflowFloat, colour toggle: NOT FuncModule_RS485_MFC.serialConnected
    Rectangle (162,397 50x27), "%d", text variable: gICP.MFC7.setFlow, colour toggle: gICP.MFC7.setdone
        OnMouseClick: write the text variable via Default
    Rectangle (215,397 23x27), "√", colour toggle: gICP.MFC7.setbusy
        OnMouseClick: write the text variable via Default
        OnMouseClick: execute { gICP.MFC7.MFCHMItif.set:=TRUE; }
    Rectangle (241,397 18x27), "×", colour toggle: gICP.MFC7.clearbusy
        OnMouseClick: write the text variable via Default
        OnMouseClick: execute { gICP.MFC7.MFCHMItif.clear:=TRUE; }
    Label (259,401 45x19), "(500)"
    Label (39,389 44x45), "7 (He)"
    Ellipse (114,401 15x15), colour toggle: gICP.GVA7Valve.extRelay
    Ellipse (337,400 15x15), colour toggle: gICP.GVB7Valve.extRelay
    Rectangle (92,118 55x31)
        tap gICP.GVA1Valve.HMIItf.singleControltemp
    Rectangle (92,164 55x31)
        tap gICP.GVA2Valve.HMIItf.singleControltemp
    Rectangle (92,211 55x31)
        tap gICP.GVA3Valve.HMIItf.singleControltemp
    Rectangle (92,258 55x31)
        tap gICP.GVA4Valve.HMIItf.singleControltemp
    Rectangle (92,300 55x31)
        tap gICP.GVA5Valve.HMIItf.singleControltemp
    Rectangle (92,346 55x31)
        tap gICP.GVA6Valve.HMIItf.singleControltemp
    Rectangle (92,392 55x31)
        tap gICP.GVA7Valve.HMIItf.singleControltemp
    Rectangle (92,442 55x31)
        tap gICP.GVA8Valve.HMIItf.singleControltemp
    Rectangle (92,492 55x31)
        tap gICP.GVA9Valve.HMIItf.singleControltemp
    Rectangle (92,543 55x31)
        tap gICP.GV20Valve_Main.HMIItf.singleControltemp
    Rectangle (316,119 55x31)
        tap gICP.GVB1Valve.HMIItf.singleControltemp
    Rectangle (316,165 55x31)
        tap gICP.GVB2Valve.HMIItf.singleControltemp
    Rectangle (316,212 55x31)
        tap gICP.GVB3Valve.HMIItf.singleControltemp
    Rectangle (316,257 55x31)
        tap gICP.GVB4Valve.HMIItf.singleControltemp
    Rectangle (316,301 55x31)
        tap gICP.GVB5Valve.HMIItf.singleControltemp
    Rectangle (316,347 55x31)
        tap gICP.GVB6Valve.HMIItf.singleControltemp
    Rectangle (316,393 55x31)
        tap gICP.GVB7Valve.HMIItf.singleControltemp
    Rectangle (316,443 55x31)
        tap gICP.GVB8Valve.HMIItf.singleControltemp
    Rectangle (316,491 55x31)
        tap gICP.GVB9Valve.HMIItf.singleControltemp
    RoundedRectangle (725,11 234x381), colour toggle: gICP.PDV.error
    Label (747,20 192x43), "PV"
    RoundedRectangle (735,66 215x37)
    RockerSwitch (859,74 51x23), variable: gICP.PDV.HMIItf.open, behaviour: TOGGLE, style: Switch-RockerSwitch-Blue
    Ellipse (918,72 23x25), colour toggle: gICP.PDVOpenSensor
    Label (743,74 117x22), "OPEN"
    RoundedRectangle (735,111 215x37)
    RockerSwitch (859,120 52x24), variable: gICP.PDV.HMIItf.close, behaviour: TOGGLE, style: Switch-RockerSwitch-Blue
    Ellipse (918,117 23x25), colour toggle: gICP.PDVCloseSensor
    Label (743,120 117x22), "CLOSE"
    RoundedRectangle (735,156 215x37)
    Label (743,164 69x22), "MODE"
    RoundedRectangle (735,202 215x37)
    Label (743,210 87x22), "PV POS."
    RoundedRectangle (735,248 215x37)
    Label (743,256 87x22), "PV PRE."
    RoundedRectangle (735,294 215x37)
    Label (743,302 106x22), "SET POINT"
    Rectangle (855,299 38x28), "%.1f", text variable: gICP.PDV.HMIItf.setPressure, colour toggle: gICP.PDV.HMIItf.setPointNotEq, input disabled if: gICP.PDV.error
        OnMouseClick: write the text variable via Default
    RockerSwitch (859,164 52x24), variable: gICP.PDV.HMIItf.mode, behaviour: TOGGLE, style: Switch-RockerSwitch-Blue
    RoundedRectangle (813,164 36x21), "PRE.", colour toggle: gICP.PDVModeRelay
    RoundedRectangle (910,164 36x21), "POS.", colour toggle: gICP.PDVModeRelay
    Label (911,209 23x22), "%"
    RoundedRectangle (855,206 38x28), "%.1f", text variable: gICP.PDV.actPos
    RoundedRectangle (855,252 38x28), "%.1f", text variable: gICP.PDV.actPressure
    Label (900,256 47x22), "mTorr"
    Rectangle (897,299 22x28), "√", colour toggle: gICP.PDV.HMIItf.setflag, input disabled if: gICP.PDV.error
        OnMouseClick: write the text variable via Default
        OnMouseClick: execute { gICP.PDV.HMIItf.set:=true; }
    Rectangle (922,299 18x28), "×", colour toggle: gICP.PDV.HMIItf.clearflag, input disabled if: gICP.PDV.error
        OnMouseClick: write the text variable via Default
        OnMouseClick: execute { gICP.PDV.HMIItf.clear:=true; }
    Rectangle (857,158 55x30), input disabled if: gICP.PDV.error
        tap gICP.PDV.HMIItf.modetemp
    Rectangle (857,115 55x31)
        tap gICP.PDV.HMIItf.closetemp
    Rectangle (852,69 62x30)
        tap gICP.PDV.HMIItf.opentemp
    RoundedRectangle (484,11 234x381), colour toggle: Not FuncModule_RS232_TBP.serialConnected
    Label (506,20 192x43), "TURBO PUM"
    RoundedRectangle (494,66 215x37)
    Ellipse (677,72 23x25), colour toggle: gICP.TruboPumOpen
    Label (499,75 67x22), "START"
    RoundedRectangle (494,111 215x37)
    RoundedRectangle (494,203 215x37)
    Ellipse (677,162 23x25), colour toggle: gICP.TruboPumNormal
    Label (502,164 117x22), "NORMAL"
    RoundedRectangle (494,157 215x37)
    Ellipse (677,117 23x25), colour toggle: gICP.TruboPumAcc
    Label (502,119 140x22), "ACCELERATE"
    RoundedRectangle (494,249 215x37)
    Ellipse (677,209 23x25), colour toggle: gICP.TruboPumDcc
    Label (502,210 117x22), "BRACK"
    RoundedRectangle (494,295 215x37)
    Ellipse (677,254 23x25), colour toggle: gICP.TruboPumError
    Label (502,256 117x22), "FAILURE"
    RoundedRectangle (494,341 215x37)
    Label (502,349 70x22), "SPEED"
    Label (666,351 31x22), "HZ"
    RoundedRectangle (604,346 56x28), "%d", text variable: gICP.TruboPumRotationSpeed
    Label (622,75 57x22), "STOP"
    RockerSwitch (566,75 53x22), variable: gICP.TruboPum.HMIItf.singleControl, behaviour: TOGGLE, style: Switch-RockerSwitch-Blue
    Label (502,303 105x22), "Temp."
    Label (666,305 31x22), "℃"
    RoundedRectangle (604,300 56x28), "%.1f", text variable: gICP.TruboPumTMS
    Rectangle (564,70 55x31)
        tap gICP.TruboPum.HMIItf.singleControltemp
    RoundedRectangle (651,724 232x129)
    RoundedRectangle (658,781 221x24)
    Label (692,728 162x23), "CHILLER"
    RoundedRectangle (658,753 221x24)
    Label (665,758 49x16), "T1"
    RoundedRectangle (713,755 32x20), "%.1f", text variable: gICP.Chiller.RTD1, colour toggle: gICP.Chiller.Error
    Label (751,759 14x15), "℃"
    RockerSwitch (739,785 45x18), variable: gICP.Chiller.HMIItf.singleControl, behaviour: TOGGLE, style: Switch-RockerSwitch-Blue
    Ellipse (853,785 19x18), colour toggle: gICP.Chiller.extRelay
    Label (664,785 70x18), "START"
    Label (781,785 59x18), "STOP"
    RoundedRectangle (658,812 221x28)
    Label (666,816 89x18), "SET POINT"
    Rectangle (787,814 49x23), "%.1f", text variable: gICP.Chiller.setpointVal
        OnMouseClick: write the text variable via Default
    Rectangle (852,814 19x23), "√", colour toggle: gICP.Chiller.busy and gICP.Chiller.setStep<>0
        OnMouseClick: write the text variable via Default
        OnMouseClick: execute { gICP.Chiller.HMIItf.set:=TRUE; }
    Label (857,759 14x15), "℃"
    Label (772,758 49x16), "T2"
    RoundedRectangle (820,755 32x20), "%.1f", text variable: gICP.Chiller.RTD2, colour toggle: gICP.Chiller.Error
    Rectangle (734,780 52x26)
        tap gICP.Chiller.HMIItf.singleControltemp
    Group (8,625 484x226), input disabled if: gWarmShowHMI.showFlag
        RoundedRectangle (0,0 484x226)
        Label (30,1 423x42), "DRY PUM"
        RoundedRectangle (12,43 221x36)
        Ellipse (200,49 24x24), colour toggle: gICP.MachianicalPumOpen
        Label (21,51 172x21), "START"
        RoundedRectangle (248,43 221x36)
        Label (256,51 77x21), "ACC"
        RoundedRectangle (248,178 221x36)
        Label (256,186 97x22), "SPEED"
        Ellipse (438,49 24x24), colour toggle: gICP.MachianicalPum.Accing
        RockerSwitch (142,52 53x23), variable: gICP.MachianicalPum.HMIItf.singleControl, behaviour: TOGGLE, style: Switch-RockerSwitch-Blue
        RoundedRectangle (371,182 68x27), "%s", text variable: gICP.MachianicalPum.DryPumpSpeed
        Label (445,187 21x21), "%"
        RoundedRectangle (13,178 221x36)
        Label (22,186 134x22), "TEMP"
        RoundedRectangle (156,182 50x27), "%s", text variable: gICP.MachianicalPum.DryPumpTemperature
        Label (212,187 21x21), "℃"
        RoundedRectangle (12,88 221x36)
        Ellipse (200,94 24x24), colour toggle: gICP.MachianicalPum.Normal
        Label (21,96 100x21), "NORMAL"
        RoundedRectangle (248,88 221x36)
        Label (256,96 77x21), "BRACK"
        Ellipse (438,94 24x24), colour toggle: gICP.MachianicalPum.Dccing
        RoundedRectangle (12,132 221x36)
        Ellipse (200,138 24x24), colour toggle: gICP.MachianicalPumAlm
        Label (21,140 172x21), "FAILURE"
        RoundedRectangle (248,132 221x36)
        Label (256,140 97x22), "CURRENT"
        RoundedRectangle (371,136 68x27), "%s", text variable: gICP.MachianicalPum.DryPumpCurrent
        Label (445,141 21x21), "A"
        Rectangle (135,45 62x31)
            tap gICP.MachianicalPum.HMIItf.singleControltemp
    RoundedRectangle (499,656 152x94)
    Label (510,659 131x34), "FORELINE"
    RockerSwitch (512,689 60x25), variable: gICP.ForlinLineValve.HMIItf.singleControl, behaviour: TOGGLE, style: Switch-RockerSwitch-Blue
    Ellipse (612,691 25x25), colour toggle: gICP.ForlinLineValveExtRelay
    Label (594,719 50x22), "mTorr"
    RoundedRectangle (510,718 76x24), "%s", text variable: gICP.ForeLineGauge.outputValue_String, colour toggle: gICP.ForeLineGauge.error
    Rectangle (508,684 68x31)
        tap gICP.ForlinLineValve.HMIItf.singleControltemp
    RoundedRectangle (979,218 178x70)
    Label (981,226 177x28), "ISO.VALVE"
    RockerSwitch (1011,259 66x22), variable: gICP.ISOValve.HMIItf.singleControl, behaviour: TOGGLE, style: Switch-RockerSwitch-Blue
    Ellipse (1098,257 20x22), colour toggle: gICP.ISOExtRelay
    Rectangle (1011,255 60x27)
        tap gICP.ISOValve.HMIItf.singleControltemp
    Group (1233,224 251x244), input disabled if: gWarmShowHMI.showFlag
        RoundedRectangle (0,0 251x244)
        Label (24,1 199x45), "LOAD LOCK"
        RoundedRectangle (17,49 215x39)
        Ellipse (199,55 25x25), colour toggle: gICP.I_WaferCheck
        Label (25,57 167x23), "WAFER ON ARM"
        RoundedRectangle (17,96 215x39)
        Label (25,105 117x23), "LL LID"
        RoundedRectangle (17,192 215x39)
        Label (25,201 94x24), "PRE."
        RoundedRectangle (17,144 215x39)
        Ellipse (199,151 25x25), colour toggle: gICP.VentExtRelay
        Label (25,153 140x23), "LL VENT"
        RoundedRectangle (150,100 73x29), "%s", text variable: gICP.I_LLSwitchString
        RockerSwitch (145,153 52x25), variable: gICP.VentValve.HMIItf.singleControl, behaviour: TOGGLE, style: Switch-RockerSwitch-Blue
        RoundedRectangle (120,196 66x29), "%s", text variable: gICP.LoadLockGauge.outputValue_String, colour toggle: gICP.LoadLockGauge.error
        Label (186,202 48x23), "mTorr"
        Rectangle (137,146 60x31)
            tap gICP.VentValve.HMIItf.singleControltemp
    Group (1224,556 178x74), input disabled if: gWarmShowHMI.showFlag
        RoundedRectangle (0,0 178x74)
        Label (5,3 162x32), "GATE DOOR"
        RockerSwitch (58,39 60x25), variable: gICP.GateDoorValve.HMIItf.singleControl, behaviour: TOGGLE, style: Switch-RockerSwitch-Blue
        RoundedRectangle (127,40 36x21), "Close", colour toggle: gICP.GateDoorRetSensor
        RoundedRectangle (14,40 36x21), "Open", colour toggle: gICP.GateDoorExtSensor
        Rectangle (55,34 65x31)
            tap gICP.GateDoorValve.HMIItf.singleControltemp
    Group (1182,672 227x107), input disabled if: gWarmShowHMI.showFlag
        RoundedRectangle (118,0 109x107)
        Label (128,4 93x63), "FAST VALVE"
        RockerSwitch (129,73 60x25), variable: gICP.FastPummingValve.HMIItf.singleControl, behaviour: TOGGLE, style: Switch-RockerSwitch-Blue
        Ellipse (197,71 25x25), colour toggle: gICP.FastPummingExtRelay
        RoundedRectangle (0,0 109x107)
        Label (10,4 93x63), "SLOW VALVE"
        RockerSwitch (11,73 60x25), variable: gICP.SlowPummingValve.HMIItf.singleControl, behaviour: TOGGLE, style: Switch-RockerSwitch-Blue
        Ellipse (79,71 25x25), colour toggle: gICP.SlowPummingExtRelay
        Rectangle (8,69 65x31)
            tap gICP.SlowPummingValve.HMIItf.singleControltemp
        Rectangle (126,69 65x31)
            tap gICP.FastPummingValve.HMIItf.singleControltemp
    RoundedRectangle (1493,367 250x347), colour toggle: gICP.PowerRF.error
    Label (1517,370 192x47), "POWER RF"
    RoundedRectangle (1505,414 225x40)
    RockerSwitch (1631,424 52x22), variable: gICP.PowerRF.openRelay, behaviour: TOGGLE, style: Switch-RockerSwitch-Blue
    Ellipse (1695,420 25x26), colour toggle: gICP.PowerRFOpenRelay
    Label (1513,422 117x23), "POWER"
    RoundedRectangle (1505,562 225x40)
    RoundedRectangle (1505,611 225x40)
    RoundedRectangle (1505,660 225x40)
    RoundedRectangle (1505,463 225x40)
    Label (1512,474 111x22), "SET POINT"
    Rectangle (1632,470 38x29), "%d", text variable: gICP.PowerRF.HMIItf.setpower, colour toggle: gICP.PowerRF.HMIItf.setpower<>gICP.PowerRF.setpower or gICP.PowerRF.setpower<>gICP.PowerRF.setpowerRead, input disabled if: S_CO_ControlRF.busy
        OnMouseClick: write the text variable via Default
    Rectangle (1678,470 23x29), "√", input disabled if: S_CO_ControlRF.busy
        OnMouseClick: write the text variable via Default
        OnMouseClick: execute { gICP.PowerRF.setpower:=gICP.PowerRF.HMIItf.setpower; gICP.PowerRF.Act_Write(); }
    Rectangle (1704,470 18x29), "×", input disabled if: S_CO_ControlRF.busy
        OnMouseClick: write the text variable via Default
        OnMouseClick: execute {
            gICP.PowerRF.setpower:=0;
            gICP.PowerRF.HMIItf.setpower:=0;
            gICP.PowerRF.Act_Write();
        }
    RoundedRectangle (1505,512 225x40)
    Label (1512,524 111x22), "TIME"
    Rectangle (1632,520 38x29), "%d", text variable: gICP.PowerRF.HMIItf.settime, colour toggle: gICP.PowerRF.HMIItf.settime<>gICP.PowerRF.settime
        OnMouseClick: write the text variable via Default
    Rectangle (1678,520 23x29), "√"
        OnMouseClick: write the text variable via Default
        OnMouseClick: execute { gICP.PowerRF.settime:=gICP.PowerRF.HMIItf.settime; }
    Rectangle (1704,520 18x29), "×"
        OnMouseClick: write the text variable via Default
        OnMouseClick: execute { gICP.PowerRF.settime:=0; gICP.PowerRF.HMIItf.settime:=0; }
    Label (1512,573 155x22), "REM. TIME"
    RoundedRectangle (1670,568 38x29), "%d", text variable: gICP.PowerRF.rematime, colour toggle: gICP.PowerRF.rematime<>0
    Label (1710,573 16x22), "S"
    Label (1512,620 155x22), "REF. POWER"
    RoundedRectangle (1669,616 38x29), "%d", text variable: gICP.PowerRF.reflectedpower, colour toggle: gICP.PowerRF.reflectedpower<>0
    Label (1709,620 16x22), "W"
    Label (1512,670 155x22), "FOR. POWER"
    RoundedRectangle (1669,666 38x29), "%d", text variable: gICP.PowerRF.forwardpower, colour toggle: (gICP.PowerRF.openbusy AND ABS(gICP.PowerRF.forwardpower-gICP.PowerRF.setpower)>2) OR (not gICP.PowerRF.busy and gICP.PowerRF.forwardpower>0) OR (gICP.PowerRF.closebusy and gICP.PowerRF.forwardpower>0)
    Label (1709,670 16x22), "W"
    Rectangle (1624,419 65x31), input disabled if: S_CO_ControlRF.busy
        tap gICP.PowerRF.HMIItf.singleControltemp
    RoundedRectangle (979,11 234x157)
    Label (1001,20 192x42), "AIM GAUGE"
    RoundedRectangle (989,64 215x36)
    RockerSwitch (1113,72 52x23), variable: gICP.AIMValve.HMIItf.singleControl, behaviour: TOGGLE, style: Switch-RockerSwitch-Blue
    Ellipse (1172,70 25x25), colour toggle: gICP .AIMExtRelay
    Label (997,72 117x21), "ENABLE"
    RoundedRectangle (989,108 215x36)
    Label (997,117 90x21), "PRE."
    RoundedRectangle (1090,113 78x27), "%s", text variable: gICP.AIMGauge.outputValue_String, colour toggle: gICP.AIMGauge.error
    Label (1168,117 34x21), "Torr"
    Rectangle (1106,66 65x31)
        tap gICP.AIMValve.HMIItf.singleControltemp
    RoundedRectangle (881,664 85x81)
    Label (883,668 82x49), "ROUGH VALVE"
    RockerSwitch (886,720 43x20), variable: gICP.RoughValve.HMIItf.singleControl, behaviour: TOGGLE, style: Switch-RockerSwitch-Blue
    Ellipse (936,715 25x25), colour toggle: gICP.RoughValveExtRelay
    Rectangle (882,714 52x26)
        tap gICP.RoughValve.HMIItf.singleControltemp
    Button (49,27 56x23), "GVA ALL OP", colour toggle: gICP.S_GASBOX_AllGVAOpen
        tap gICP.C_GASBOX_AllGVAOpenTemp
    Button (112,27 56x23), "GVA ALL CL", colour toggle: gICP.S_GASBOX_AllGVAClose
        tap gICP.C_GASBOX_AllGVACloseTemp
    Button (387,27 56x23), "GVB ALL CL", colour toggle: gICP.S_GASBOX_AllGVBClose
        tap gICP.C_GASBOX_AllGVBCloseTemp
    Button (324,27 56x23), "GVB ALL OP", colour toggle: gICP.S_GASBOX_AllGVBOpen
        tap gICP.C_GASBOX_AllGVBOpenTemp
    Button (157,87 48x23), "ALL Set"
        tap gICP.C_GASBOX_AllMFCSetTemp
    Button (256,87 48x23), "ALL Clear"
        tap gICP.C_GASBOX_AllMFCClearTemp
    RoundedRectangle (1493,11 250x350), colour toggle: gICP.SourceRF.error
    Label (1518,14 192x47), "SOURCE RF"
    RoundedRectangle (1505,58 225x40)
    RockerSwitch (1631,68 52x22), variable: gICP.SourceRF.openRelay, behaviour: TOGGLE, style: Switch-RockerSwitch-Blue
    Ellipse (1695,64 25x26), colour toggle: gICP.SourceRFOpenRelay
    Label (1513,66 117x23), "POWER"
    RoundedRectangle (1505,206 225x40)
    RoundedRectangle (1505,255 225x40)
    RoundedRectangle (1505,304 225x40)
    RoundedRectangle (1505,107 225x40)
    Label (1512,118 111x22), "SET POINT"
    Rectangle (1632,114 38x29), "%d", text variable: gICP.SourceRF.HMIItf.setpower, colour toggle: gICP.SourceRF.HMIItf.setpower<>gICP.SourceRF.setpower or gICP.SourceRF.setpower<>gICP.SourceRF.setpowerRead, input disabled if: S_CO_ControlRF.busy
        OnMouseClick: write the text variable via Default
    Rectangle (1678,114 23x29), "√", input disabled if: S_CO_ControlRF.busy
        OnMouseClick: write the text variable via Default
        OnMouseClick: execute { gICP.SourceRF.setpower:=gICP.SourceRF.HMIItf.setpower; gICP.SourceRF.Act_Write(); }
    Rectangle (1704,114 18x29), "×", input disabled if: S_CO_ControlRF.busy
        OnMouseClick: write the text variable via Default
        OnMouseClick: execute {
            gICP.SourceRF.setpower:=0;
            gICP.SourceRF.HMIItf.setpower:=0;
            gICP.SourceRF.Act_Write();
        }
    RoundedRectangle (1505,156 225x40)
    Label (1512,168 111x22), "TIME"
    Rectangle (1632,164 38x29), "%d", text variable: gICP.SourceRF.HMIItf.settime, colour toggle: gICP.SourceRF.HMIItf.settime<>gICP.SourceRF.settime
        OnMouseClick: write the text variable via Default
    Rectangle (1678,164 23x29), "√"
        OnMouseClick: write the text variable via Default
        OnMouseClick: execute { gICP.SourceRF.settime:=gICP.SourceRF.HMIItf.settime; }
    Rectangle (1704,164 18x29), "×"
        OnMouseClick: write the text variable via Default
        OnMouseClick: execute { gICP.SourceRF.settime:=0; gICP.SourceRF.HMIItf.settime:=0; }
    Label (1512,217 155x22), "REM. TIME"
    RoundedRectangle (1670,212 38x29), "%d", text variable: gICP.SourceRF.rematime, colour toggle: gICP.SourceRF.rematime<>0
    Label (1710,217 16x22), "S"
    Label (1512,264 155x22), "REF. POWER"
    RoundedRectangle (1669,260 38x29), "%d", text variable: gICP.SourceRF.reflectedpower, colour toggle: gICP.SourceRF.reflectedpower<>0
    Label (1709,264 16x22), "W"
    Label (1512,314 155x22), "FOR. POWER"
    RoundedRectangle (1669,310 38x29), "%d", text variable: gICP.SourceRF.forwardpower, colour toggle: (gICP.SourceRF.openbusy AND ABS(gICP.SourceRF.forwardpower-gICP.SourceRF.setpower)>2) OR (not gICP.SourceRF.busy and gICP.SourceRF.forwardpower>0)
    Label (1709,314 16x22), "W"
    Rectangle (1623,63 65x31), input disabled if: S_CO_ControlRF.busy
        tap gICP.SourceRF.HMIItf.singleControltemp
    RoundedRectangle (1401,147 61x29), "%d", text variable: gICP.ARM.actpos
    Rectangle (1251,18 64x29), "P:%d", text variable: gARMPosition
        OnMouseClick: write the text variable via Default, min 0, max 9000
    Rectangle (1409,18 55x29), "V:%d", text variable: gICP.ARM.setvel
        OnMouseClick: write the text variable via Default, min 1, max 30
    Rectangle (1357,103 37x29), "L:%d", text variable: gICP.ARM.jogsetlen
        OnMouseClick: write the text variable via Default, min 1, max 10
    RoundedRectangle (1353,152 45x21), "STOP", input disabled if: NOT FuncModule_RS232_ARM.serialConnected
        OnMouseClick: write the text variable via Default
        OnMouseClick: execute { gICP.ARM.Act_Stop(); }
    Line (308,582) (455,582)
    Label (386,539 61x42), "GVA10 (Vent)"
    RockerSwitch (319,548 53x23), variable: gICP.GVA10Valve_Vent.HMIItf.singleControl, behaviour: TOGGLE, style: Switch-RockerSwitch-Blue
    Ellipse (338,551 15x15), colour toggle: gICP.GVA10Valve_Vent.extRelay
    Rectangle (316,543 55x31)
        tap gICP.GVA10Valve_Vent.HMIItf.singleControltemp
    RoundedRectangle (1430,720 312x132)
    Label (1488,723 192x36), "RF Co-Control"
    RoundedRectangle (1551,802 181x40)
    Label (1556,811 97x22), "REM. TIME"
    RoundedRectangle (1657,808 38x29), "%d", text variable: gCO_ControlRFRMTime, colour toggle: gCO_ControlRFRMTime>1
    Label (1701,811 16x22), "S"
    RoundedRectangle (1551,758 180x40)
    Label (1556,768 96x22), "SET TIME"
    Rectangle (1657,764 38x29), "%d", text variable: gCO_ControlRFTime
        OnMouseClick: write the text variable via Default
    RoundedRectangle (1439,758 107x85)
    RoundedRectangle (1450,765 51x27), "START", input disabled if: NOT(gICP.PowerRF.openCondition AND gICP.SourceRF.openCondition) OR S_CO_ControlRF.busy
        OnMouseClick: write the text variable via Default
        OnMouseClick: execute {
            S_CO_ControlRF.Act_Init_Status();
            S_CO_ControlRF.Act_Ex();
            S_CO_ControlRF.bTrig:=TRUE;
        }
    Ellipse (1511,766 25x26), colour toggle: S_CO_ControlRF.busy
    RoundedRectangle (1450,805 51x27), "STOP"
        OnMouseClick: write the text variable via Default
        OnMouseClick: execute { S_CO_ControlRF.bStop:=TRUE; S_CO_ControlRF.bAbort:=TRUE; }
    Ellipse (1511,806 25x26), colour toggle: S_CO_ControlRF.stopDone
    Rectangle (896,791 52x26)
        tap gICP.RoughValve.HMIItf.singleControltemp
    RoundedRectangle (896,788 510x66)
    Label (905,789 186x34), "BACK OF HELIUM"
    RoundedRectangle (907,824 97x26)
    RockerSwitch (934,829 44x20), variable: gICP.HeINValve.HMIItf.singleControl, behaviour: TOGGLE, style: Switch-RockerSwitch-Blue
    Ellipse (980,827 21x20), colour toggle: gICP.HeINExtRelay
    Label (909,827 25x21), "HI"
    RoundedRectangle (1010,824 106x26)
    RockerSwitch (1046,829 44x20), variable: gICP.HePumValve.HMIItf.singleControl, behaviour: TOGGLE, style: Switch-RockerSwitch-Blue
    Ellipse (1092,827 21x20), colour toggle: gICP.HePumExtRelay
    Label (1012,827 32x21), "HO"
    RoundedRectangle (1123,793 271x26)
    Label (1126,796 32x21), "PRE"
    RoundedRectangle (1121,824 274x26)
    Label (1127,827 32x21), "MFC"
    Label (1234,795 41x22), "Torr"
    RoundedRectangle (1164,796 67x20), "%.3f", text variable: gICP.HeCheckGaugeReal
    RoundedRectangle (1275,827 68x20), "%.1f", text variable: gICP.HeMFC_ActFlow
    Label (1345,827 44x22), "Sccm"
    Rectangle (934,824 41x26)
        tap gICP.HeINValve.HMIItf.singleControltemp
    Rectangle (1046,824 41x26)
        tap gICP.HePumValve.HMIItf.singleControltemp
    Ellipse (1026,505 120x2), colour toggle: gWaferMemoryState=1
        OnMouseClick: execute { gWaferMemoryState:=BOOL_TO_INT(NOT INT_TO_BOOL(gWaferMemoryState)); ups_CX51X0.Act_Wrtie(); }
    Label (988,442 177x32), "Wafer In Chamber", invisible if: NOT otherMachineState.lightShow
    Label (965,399 230x32), "Chamber ATM state", invisible if: NOT gICP.I_ATMSensor
    RoundedRectangle (979,295 177x58)
    Label (994,300 150x26), "Chamber"
    Label (1096,326 50x22), "mTorr"
    RoundedRectangle (998,325 89x24), "%.1f", text variable: gICP.ChamberGauge.outputValue1, colour toggle: gICP.ChamberGauge.error
    Rectangle (1163,827 68x20), "Set:%.1f", text variable: gICP.HeMFC_SetFlowHMI
        OnMouseClick: write the text variable via Default, min 0, max 100
    Label (1233,826 41x22), "Sccm"
    RoundedRectangle (485,400 234x67)
    Label (496,405 212x26), "TURBO PUM TAIL"
    Label (651,434 50x22), "mTorr"
    RoundedRectangle (504,433 104x24), "%.1f", text variable: gICP.TBGauge.outputValue, colour toggle: gICP.TBGauge.error
    RoundedRectangle (1348,795 41x21), "record", colour toggle: MainRunPOU.testLog
        toggle MainRunPOU.testLog
        OnMouseClick: write the text variable via Default
END_VISUALIZATION

// ---- VISUs/Config/Config.TcVIS
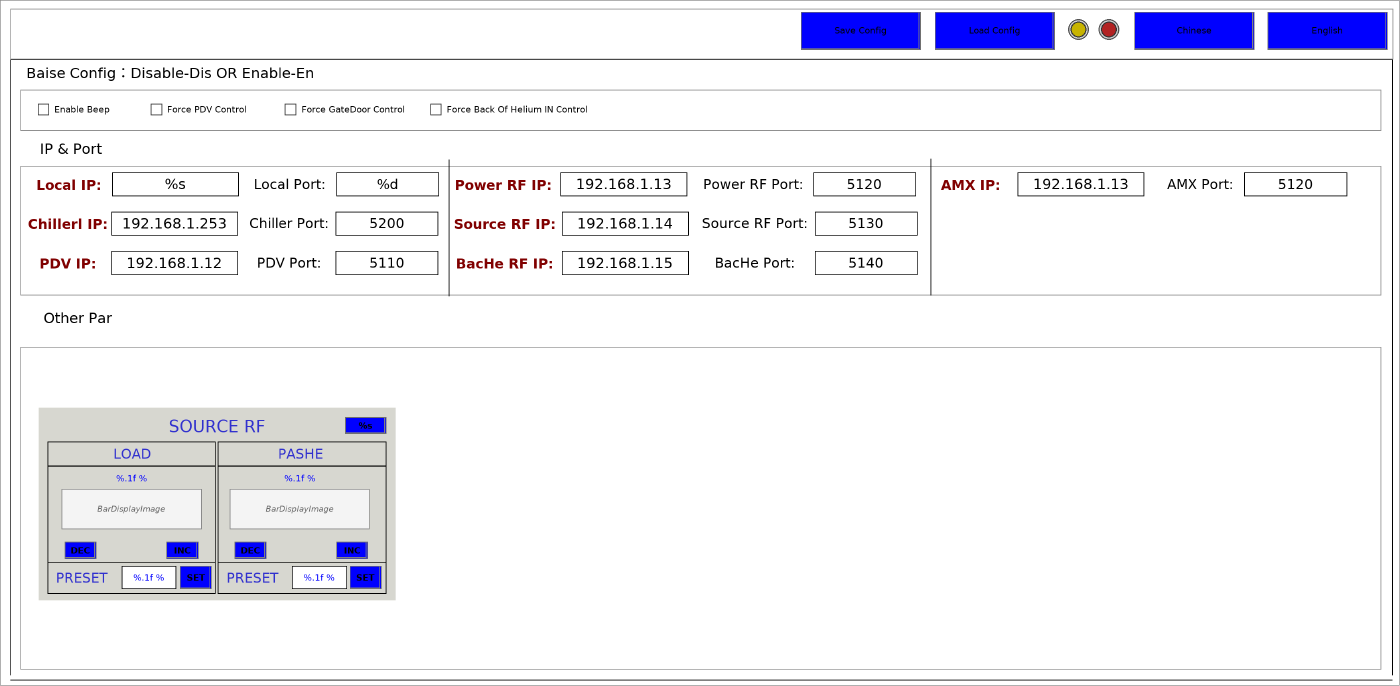
VISUALIZATION Config  // 1755x860
    Frame (13,74 1732x780), input disabled if: gAutoRunningFlag OR gRunningState=RunningStatus.eHomeState
        shows Config_Base()
        shows DataView()
        shows Config_TestSocket()
        shows Config_TXTest()
        shows Config_Coaxial()
        shows Config_RXTest()
        shows Config_UnLoad()
    GroupBox (13,3 1733x71)
        Button (1409,12 150x47), "Chinese"
            OnMouseUp: ChangeLanguage ChangeLanguage=Chinese
            OnMouseUp: execute { gCNErrShow:=TRUE; }
        Button (1576,12 150x47), "English"
            OnMouseUp: ChangeLanguage ChangeLanguage=English
            OnMouseUp: execute { gCNErrShow:=FALSE; }
        Button (1159,12 150x47), "Load Config"
            tap gRead
        Button (991,12 150x47), "Save Config"
            tap gSave
        Lamp1 (1324,19 30x30), variable: DataSave.busy, style: Lamp-Lamp1-Yellow
        Lamp1 (1362,19 30x30), variable: DataSave.error or FB_WStringSave.readError or FB_WStringSave.saveError, style: Lamp-Lamp1-Red
END_VISUALIZATION

// ---- VISUs/Config/Config_Base.TcVIS
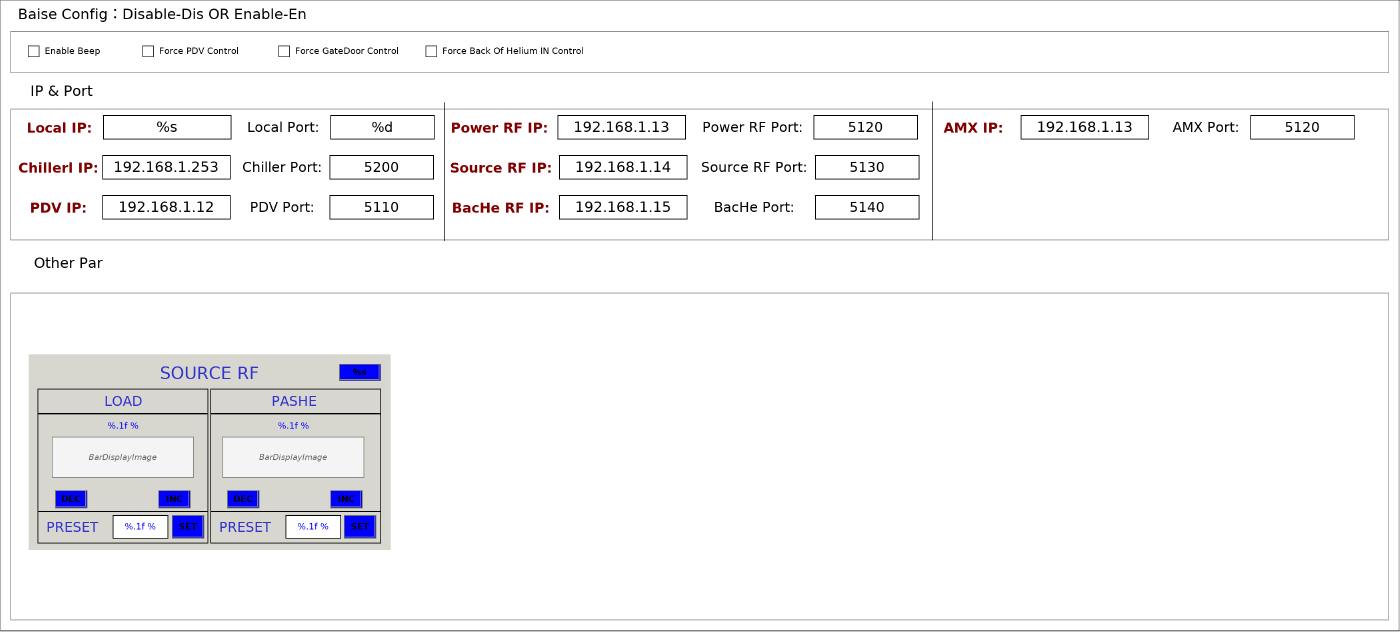
VISUALIZATION Config_Base  // 1750x790
    Group (0,0 1751x0)
        Line (0,788) (1750,788)
        Line (0,0) (0,782)
        Line (0,0) (1750,0)
        Line (1750,0) (1750,782)
    GroupBox (13,358 1723x417)
        Label (-2382,-64 501x61), "参数设置说明"
        Label (-2397,-19 522x195), "需切换界面左上角控制模式为“配置模式”，根据参数栏 左上方提示内容及其设置框说明标题，设置相应的参数并按 “保存配置”按钮3秒以上，直到右侧黄灯闪烁 设置完成参数后需根据相应需求选择对应控制模式"
        RoundedRectangle (23,85 452x244), colour toggle: NOT FuncModule_RS232_SRF.serialConnected
        Rectangle (250,159 213x162)
        Rectangle (34,159 213x162)
        Label (153,93 192x31), "SOURCE RF"
        RoundedRectangle (34,281 213x40)
        Label (42,290 85x22), "PRESET"
        RoundedRectangle (128,286 69x29), "%.1f %", text variable: FuncModule_RS232_SRF.goPosLoad, input disabled if: TRUE
            OnMouseClick: write the text variable via Default, min 0.0, max 100.0
        Button (56,255 40x22), "DEC", input disabled if: TRUE
            OnMouseClick: execute { FuncModule_RS232_SRF.LoadDEC(); }
        Button (185,255 40x22), "INC", input disabled if: TRUE
            OnMouseClick: execute { FuncModule_RS232_SRF.LoadINC(); }
        Button (271,255 40x22), "DEC", input disabled if: TRUE
            OnMouseClick: execute { FuncModule_RS232_SRF.PhaseDEC(); }
        Button (400,255 40x22), "INC", input disabled if: TRUE
            OnMouseClick: execute { FuncModule_RS232_SRF.PhaseINC(); }
        Button (202,286 40x29), "SET", input disabled if: TRUE
            OnMouseClick: execute { FuncModule_RS232_SRF.LoadAndPhaseGo(); }
        RoundedRectangle (250,281 213x40)
        Label (258,290 85x22), "PRESET"
        RoundedRectangle (344,286 69x29), "%.1f %", text variable: FuncModule_RS232_SRF.goPosPhase, input disabled if: TRUE
            OnMouseClick: write the text variable via Default, min 0.0, max 100.0
        Button (417,286 40x29), "SET", input disabled if: TRUE
            OnMouseClick: execute { FuncModule_RS232_SRF.LoadAndPhaseGo(); }
        Rectangle (34,128 213x31)
        Label (109,133 65x21), "LOAD"
        Rectangle (250,128 213x31)
        Label (315,133 80x21), "PASHE"
        Button (411,97 52x21), "%s", text variable: FuncModule_RS232_SRF.rec_MAStr, input disabled if: TRUE
            OnMouseClick: execute { FuncModule_RS232_SRF.ManulORAuto(); }
        BarDisplayImage (52,188 177x51), value: FuncModule_RS232_SRF.load, style: BarDisplayImage-Gray, scale format: %.1f, scale 0..100
        BarDisplayImage (265,188 177x51), value: FuncModule_RS232_SRF.phase, style: BarDisplayImage-Gray, scale format: %.1f, scale 0..100
        RoundedRectangle (113,160 56x29), "%.1f %", text variable: FuncModule_RS232_SRF.load, colour toggle: FuncModule_RS232_SRF.loadRunErr
        RoundedRectangle (326,160 56x29), "%.1f %", text variable: FuncModule_RS232_SRF.phase, colour toggle: FuncModule_RS232_SRF.phashRunErr
    Label (1928,1052 45x20)
    Label (5,3 396x30), "Baise Config：Disable-Dis OR Enable-En"
    Label (5,99 144x30), "IP & Port"
    GroupBox (13,31 1723x60)
        Label (-2382,-64 501x61), "参数设置说明"
        Label (-2397,-19 522x195), "需切换界面左上角控制模式为“配置模式”，根据参数栏 左上方提示内容及其设置框说明标题，设置相应的参数并按 “保存配置”按钮3秒以上，直到右侧黄灯闪烁 设置完成参数后需根据相应需求选择对应控制模式"
        Checkbox (20,13 116x40), "Enable Beep", variable: fbMachineState.HMI_EnableBuzzer
        Checkbox (163,13 152x40), "Force PDV Control", variable: gEnablePDVOpenClose
        Checkbox (333,13 175x40), "Force GateDoor Control", variable: gEnableGDOpenClose
        Checkbox (517,13 224x40), "Force Back Of Helium IN Control", variable: gEnableHeInOpenClose
    GroupBox (13,128 1723x172)
        Label (-2382,-64 501x61), "参数设置说明"
        Label (-2397,-19 522x195), "需切换界面左上角控制模式为“配置模式”，根据参数栏 左上方提示内容及其设置框说明标题，设置相应的参数并按 “保存配置”按钮3秒以上，直到右侧黄灯闪烁 设置完成参数后需根据相应需求选择对应控制模式"
        Label (9,16 105x32), "Local IP:"
        Rectangle (116,16 160x30), "%s", text variable: gLocalHostIp, input disabled if: NOT (gRunningState=RunningStatus.eManualState AND gCtrlMode=ControlMode.eConfig)
        Rectangle (400,16 130x30), "%d", text variable: gLocalHostPort, input disabled if: NOT (gRunningState=RunningStatus.eManualState AND gCtrlMode=ControlMode.eConfig)
        Label (287,16 108x30), "Local Port:"
        Label (8,66 105x32), "Chillerl IP:"
        Label (8,116 105x32), "PDV IP:"
        Label (541,16 141x32), "Power RF IP:"
        Label (543,66 141x32), "Source RF IP:"
        Label (543,116 141x32), "BacHe RF IP:"
        Rectangle (1550,16 130x30), "5120", text variable: gLocalHostPort, input disabled if: NOT (gRunningState=RunningStatus.eManualState AND gCtrlMode=ControlMode.eConfig)
    Label (20,311 131x36), "Other Par"
    Rectangle (128,194 160x30), "192.168.1.253", text variable: gLocalHostIp, input disabled if: NOT (gRunningState=RunningStatus.eManualState AND gCtrlMode=ControlMode.eConfig)
    Rectangle (412,194 130x30), "5200", text variable: gLocalHostPort, input disabled if: NOT (gRunningState=RunningStatus.eManualState AND gCtrlMode=ControlMode.eConfig)
    Label (299,194 108x30), "Chiller Port:"
    Rectangle (128,244 160x30), "192.168.1.12", text variable: gLocalHostIp, input disabled if: NOT (gRunningState=RunningStatus.eManualState AND gCtrlMode=ControlMode.eConfig)
    Rectangle (412,244 130x30), "5110", text variable: gLocalHostPort, input disabled if: NOT (gRunningState=RunningStatus.eManualState AND gCtrlMode=ControlMode.eConfig)
    Label (299,244 108x30), "PDV Port:"
    Rectangle (697,144 160x30), "192.168.1.13", text variable: gLocalHostIp, input disabled if: NOT (gRunningState=RunningStatus.eManualState AND gCtrlMode=ControlMode.eConfig)
    Rectangle (1017,144 130x30), "5120", text variable: gLocalHostPort, input disabled if: NOT (gRunningState=RunningStatus.eManualState AND gCtrlMode=ControlMode.eConfig)
    Label (868,144 146x30), "Power RF Port:"
    Rectangle (699,194 160x30), "192.168.1.14", text variable: gLocalHostIp, input disabled if: NOT (gRunningState=RunningStatus.eManualState AND gCtrlMode=ControlMode.eConfig)
    Rectangle (1019,194 130x30), "5130", text variable: gLocalHostPort, input disabled if: NOT (gRunningState=RunningStatus.eManualState AND gCtrlMode=ControlMode.eConfig)
    Label (870,194 146x30), "Source RF Port:"
    Rectangle (699,244 160x30), "192.168.1.15", text variable: gLocalHostIp, input disabled if: NOT (gRunningState=RunningStatus.eManualState AND gCtrlMode=ControlMode.eConfig)
    Rectangle (1019,244 130x30), "5140", text variable: gLocalHostPort, input disabled if: NOT (gRunningState=RunningStatus.eManualState AND gCtrlMode=ControlMode.eConfig)
    Label (870,244 146x30), "BacHe Port:"
    Label (1160,144 114x32), "AMX IP:"
    Rectangle (1276,144 160x30), "192.168.1.13", text variable: gLocalHostIp, input disabled if: NOT (gRunningState=RunningStatus.eManualState AND gCtrlMode=ControlMode.eConfig)
    Label (1455,144 105x30), "AMX Port:"
    Line (556,301) (556,128)
    Line (1166,300) (1166,127)
END_VISUALIZATION

// ---- VISUs/Editor/Overview_Total.TcVIS
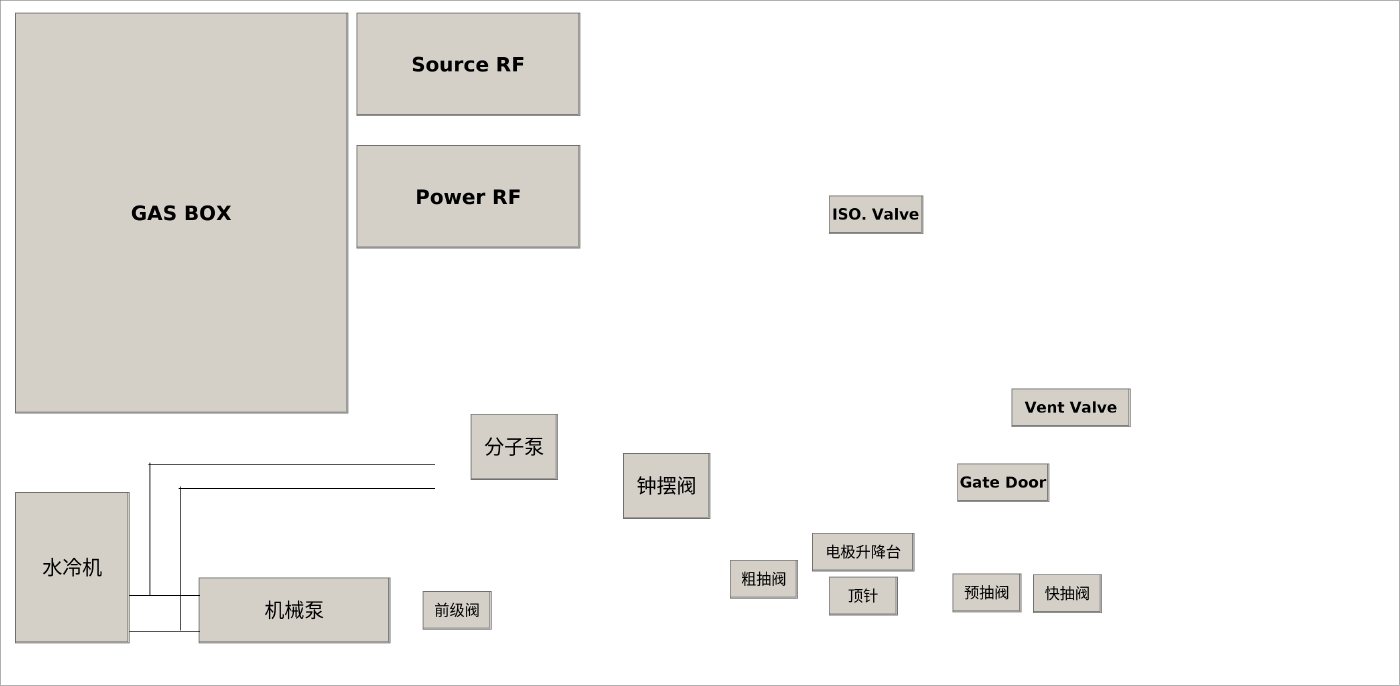
VISUALIZATION Overview_Total  // 1755x860, background image ImagePool1.autoImg
    Button (249,724 240x82), "机械泵"
    Button (19,617 143x189), "水冷机"
    Line (162,791) (250,791)
    Line (162,746) (250,746)
    Line (188,746) (188,580)
    Line (226,790) (226,610)
    Line (186,582) (545,582)
    Line (224,612) (545,612)
    Button (590,519 109x82), "分子泵"
    Button (781,568 109x82), "钟摆阀"
    Button (530,741 86x48), "前级阀"
    Button (915,702 85x48), "粗抽阀"
    Button (1018,668 128x48), "电极升降台"
    Button (1039,723 86x48), "顶针"
    Button (1194,719 86x48), "预抽阀"
    Button (1295,720 86x48), "快抽阀"
    Button (19,16 417x502), "GAS BOX"
    Button (1039,245 118x48), "ISO. Valve"
    Button (1200,581 115x48), "Gate Door"
    Button (1268,487 149x48), "Vent Valve"
    Button (447,16 280x129), "Source RF"
    Button (447,182 280x129), "Power RF"
END_VISUALIZATION

// ---- VISUs/Editor/ViewPar.TcVIS
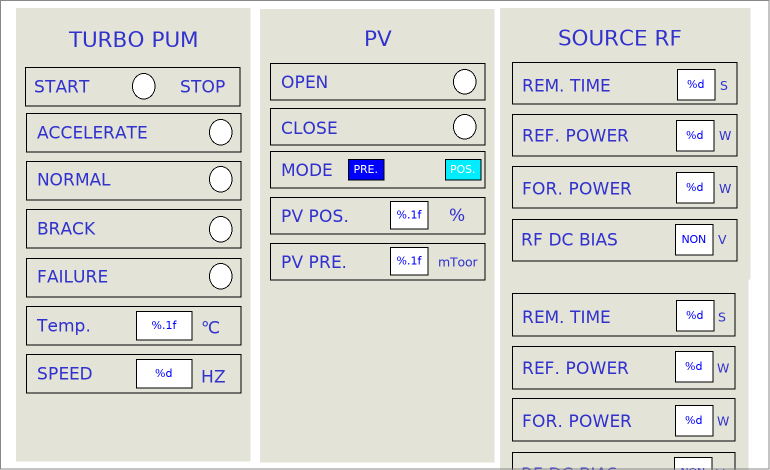
VISUALIZATION ViewPar  // 770x470
    RoundedRectangle (16,8 234x453)
    Label (38,17 192x45), "TURBO PUM"
    Ellipse (132,73 23x26), colour toggle: gICP.TruboPumOpen
    Label (31,75 67x23), "START"
    RoundedRectangle (26,113 215x39)
    RoundedRectangle (26,209 215x39)
    Ellipse (209,166 23x26), colour toggle: gICP.TruboPumNormal
    Label (34,168 117x23), "NORMAL"
    RoundedRectangle (26,161 215x39)
    Ellipse (209,119 23x26), colour toggle: gICP.TruboPumAcc
    Label (34,121 140x23), "ACCELERATE"
    RoundedRectangle (26,258 215x39)
    Ellipse (209,216 23x26), colour toggle: gICP.TruboPumDcc
    Label (34,217 117x23), "BRACK"
    RoundedRectangle (26,306 215x39)
    Ellipse (209,263 23x26), colour toggle: gICP.TruboPumError
    Label (34,265 117x23), "FAILURE"
    RoundedRectangle (26,354 215x39)
    Label (34,362 70x23), "SPEED"
    Label (198,365 31x23), "HZ"
    RoundedRectangle (136,359 56x29), "%d", text variable: gICP.TruboPumRotationSpeed
    Label (177,75 57x23), "STOP"
    Label (34,314 105x23), "Temp."
    Label (198,316 31x23), "℃"
    RoundedRectangle (136,311 56x29), "%.1f", text variable: gICP.TruboPumTMS
    RoundedRectangle (25,67 215x39)
    RoundedRectangle (260,9 234x453)
    Label (282,17 192x43), "PV"
    RoundedRectangle (270,63 215x37)
    Ellipse (453,69 23x25), colour toggle: gICP.PDVOpenSensor
    Label (278,71 117x22), "OPEN"
    RoundedRectangle (270,108 215x37)
    Ellipse (453,114 23x25), colour toggle: gICP.PDVCloseSensor
    Label (278,117 117x22), "CLOSE"
    RoundedRectangle (270,151 215x37)
    Label (278,159 69x22), "MODE"
    RoundedRectangle (270,197 215x37)
    Label (278,205 87x22), "PV POS."
    RoundedRectangle (270,243 215x37)
    Label (278,251 87x22), "PV PRE."
    RoundedRectangle (348,159 36x21), "PRE.", colour toggle: gICP.PDVModeRelay
    RoundedRectangle (445,159 36x21), "POS.", colour toggle: gICP.PDVModeRelay
    Label (446,204 23x22), "%"
    RoundedRectangle (390,201 38x28), "%.1f", text variable: gICP.PDV.actPos
    RoundedRectangle (390,247 38x28), "%.1f", text variable: gICP.PDV.actPressure
    Label (435,251 47x22), "mToor"
    Group (500,236 250x225)
        RoundedRectangle (0,0 248x276)
        Label (24,5 190x50), "POWER RF"
        RoundedRectangle (12,57 223x43)
        RoundedRectangle (12,110 223x43)
        RoundedRectangle (12,162 223x43)
        RoundedRectangle (12,216 223x43)
        Label (19,69 154x24), "REM. TIME"
        RoundedRectangle (176,64 38x31), "%d", text variable: gICP.PowerRF.rematime, colour toggle: gICP.PowerRF.rematime<>0
        Label (215,69 16x24), "S"
        Label (19,120 154x24), "REF. POWER"
        RoundedRectangle (175,115 38x31), "%d", text variable: gICP.PowerRF.reflectedpower, colour toggle: gICP.PowerRF.reflectedpower<>0
        Label (214,120 16x24), "W"
        Label (19,173 154x24), "FOR. POWER"
        RoundedRectangle (175,169 38x31), "%d", text variable: gICP.PowerRF.forwardpower, colour toggle: (gICP.PowerRF.openbusy AND ABS(gICP.PowerRF.forwardpower-gICP.PowerRF.setpower)>2) OR (not gICP.PowerRF.busy and gICP.PowerRF.forwardpower>0) OR (gICP.PowerRF.closebusy and gICP.PowerRF.forwardpower>0)
        Label (214,173 16x24), "W"
        Label (18,226 154x24), "RF DC BIAS"
        RoundedRectangle (174,221 38x31), "NON"
        Label (213,226 16x24), "V"
    Group (500,8 250x225)
        RoundedRectangle (0,0 250x271)
        Label (24,5 192x50), "SOURCE RF"
        RoundedRectangle (12,54 225x42)
        RoundedRectangle (12,106 225x42)
        RoundedRectangle (12,158 225x42)
        RoundedRectangle (12,211 225x42)
        Label (19,66 155x23), "REM. TIME"
        RoundedRectangle (177,61 38x31), "%d", text variable: gICP.SourceRF.rematime, colour toggle: gICP.SourceRF.rematime<>0
        Label (217,66 16x23), "S"
        Label (19,116 155x23), "REF. POWER"
        RoundedRectangle (176,112 38x31), "%d", text variable: gICP.SourceRF.reflectedpower, colour toggle: gICP.SourceRF.reflectedpower<>0
        Label (216,116 16x23), "W"
        Label (19,169 155x23), "FOR. POWER"
        RoundedRectangle (176,164 38x31), "%d", text variable: gICP.SourceRF.forwardpower, colour toggle: (gICP.SourceRF.busy AND ABS(gICP.SourceRF.forwardpower-gICP.SourceRF.setpower)>2) OR (not gICP.SourceRF.busy and gICP.SourceRF.forwardpower>0)
        Label (216,169 16x23), "W"
        Label (18,220 155x23), "RF DC BIAS"
        RoundedRectangle (175,216 38x31), "NON"
        Label (215,220 16x23), "V"
END_VISUALIZATION

// ---- VISUs/Editor/ViewPar_1.TcVIS
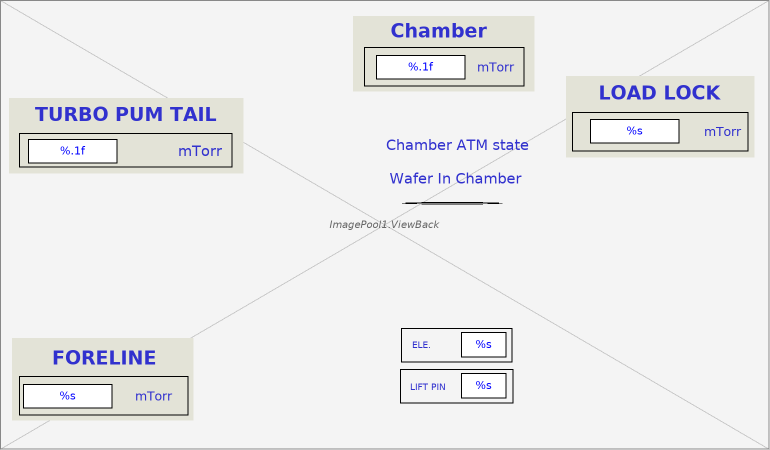
VISUALIZATION ViewPar_1  // 770x450
    Image (0,0 769x449), image: ImagePool1.ViewBack
    Label (361,129 193x32), "Chamber ATM state", invisible if: NOT gICP.I_ATMSensor
    Group (566,76 188x81)
        RoundedRectangle (0,0 188x81)
        Label (12,1 163x32), "LOAD LOCK"
        RoundedRectangle (6,36 176x39)
        RoundedRectangle (24,43 89x24), "%s", text variable: gICP.LoadLockGauge.outputValue_String, colour toggle: gICP.LoadLockGauge.error
        Label (135,44 41x23), "mTorr"
    Group (353,16 181x75)
        RoundedRectangle (0,0 181x75)
        Label (14,2 150x26), "Chamber"
        Label (121,40 50x22), "mTorr"
        RoundedRectangle (23,39 89x24), "%.1f", text variable: gICP.ChamberGauge.outputValue1, colour toggle: gICP.ForeLineGauge.error
        RoundedRectangle (11,31 160x39)
    RoundedRectangle (12,338 181x82)
    Label (39,341 131x34), "FORELINE"
    Label (132,385 50x22), "mTorr"
    RoundedRectangle (23,384 89x24), "%s", text variable: gICP.ForeLineGauge.outputValue_String, colour toggle: gICP.ForeLineGauge.error
    RoundedRectangle (19,376 169x39)
    Group (9,98 234x75)
        RoundedRectangle (0,0 234x75)
        Label (11,2 212x29), "TURBO PUM TAIL"
        Label (166,42 50x22), "mTorr"
        RoundedRectangle (19,41 89x24), "%.1f", text variable: gICP.TBGauge.outputValue, colour toggle: gICP.TBGauge.error
        RoundedRectangle (10,35 213x34)
    Ellipse (402,202 100x2), colour toggle: gWaferMemoryState=1
        OnMouseClick: execute { gWaferMemoryState:=BOOL_TO_INT(NOT INT_TO_BOOL(gWaferMemoryState)); ups_CX51X0.Act_Wrtie(); }
    Label (384,166 143x25), "Wafer In Chamber", invisible if: NOT otherMachineState.lightShow
    RoundedRectangle (401,328 111x34)
    Label (409,335 28x20), "ELE."
    RoundedRectangle (400,369 113x34)
    Label (407,377 50x20), "LIFT PIN"
    RoundedRectangle (461,332 45x25), "%s", text variable: gICP.ElectrodeCyl.HMIItf.sensorShow
    RoundedRectangle (461,373 45x25), "%s", text variable: gICP.LiftPinCyl.HMIItf.sensorShow
END_VISUALIZATION

// ---- VISUs/IO/IO.TcVIS
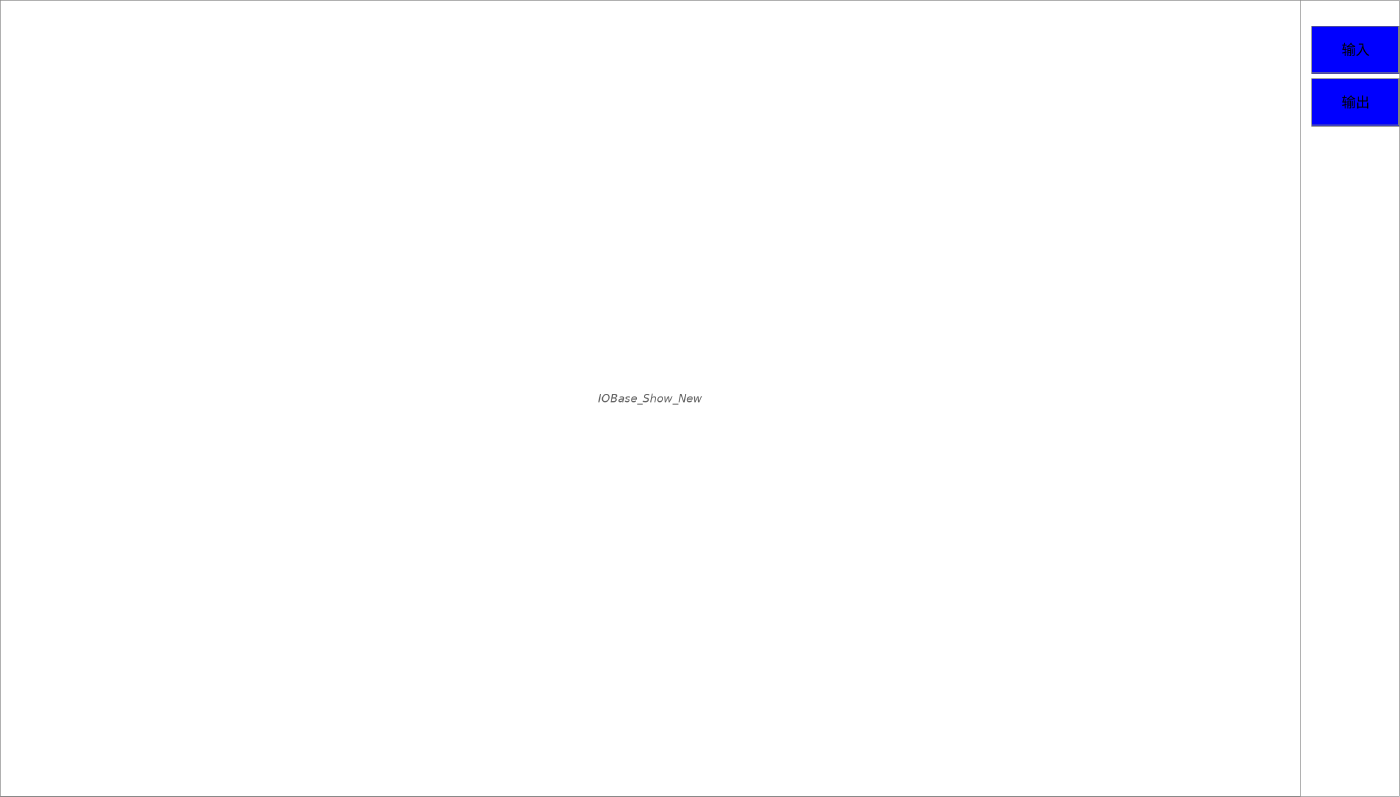
VISUALIZATION IO  // 1895x1080
    Frame (0,0 1760x1080)
        shows IO_Input()
        shows IO_Output()
        shows Auto_test_1()
    Button (1775,35 120x65), "输入"
        OnMouseClick: FrameSelectionChange Selection=SelectedFrame=1d4c33e9-a5b9-451d-bf86-00d28fadf65b, GlobSel=AssignType=Directly, SelType=Locally
    Button (1775,106 120x65), "输出"
        OnMouseClick: FrameSelectionChange Selection=SelectedFrame=1d4c33e9-a5b9-451d-bf86-00d28fadf65b, Selection=1, GlobSel=AssignType=Directly, SelType=Locally
END_VISUALIZATION

// ---- VISUs/IO/IO_Input.TcVIS
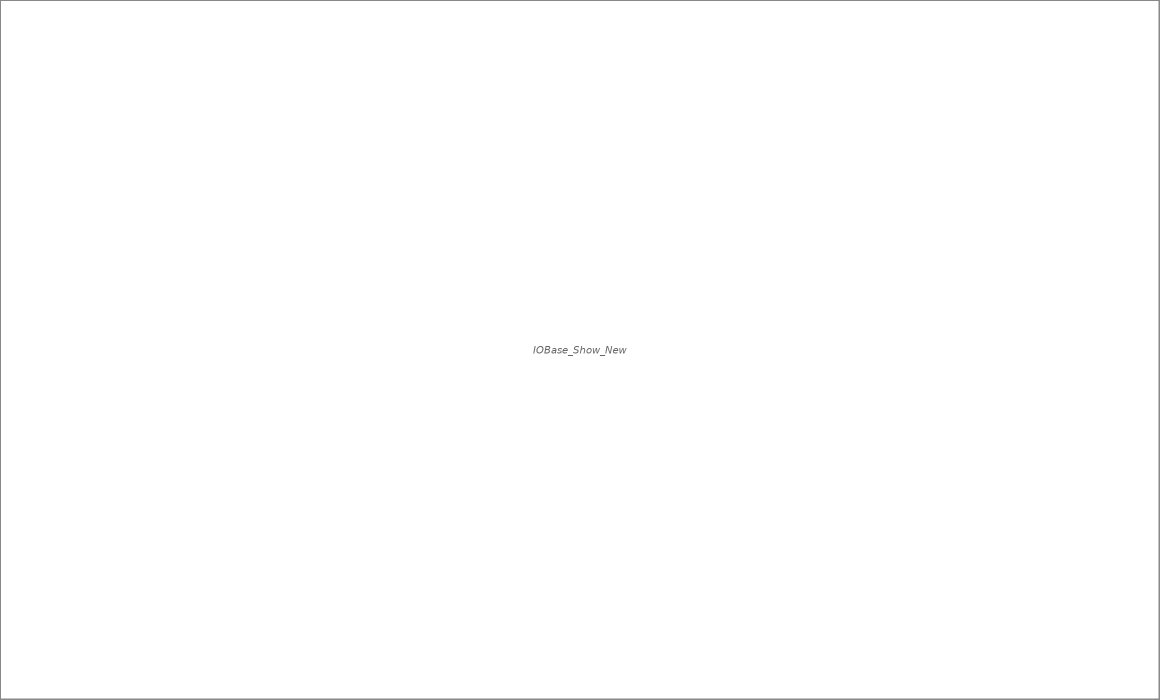
VISUALIZATION IO_Input  // 1160x700
    TabControl (0,0 1160x700)
        shows IOBase_Show_New(userData := TesterIO.fbIOBase_Input.HMIITF)
        [0]: TabTitle=Input
END_VISUALIZATION

// ---- VISUs/IO/IO_Output.TcVIS
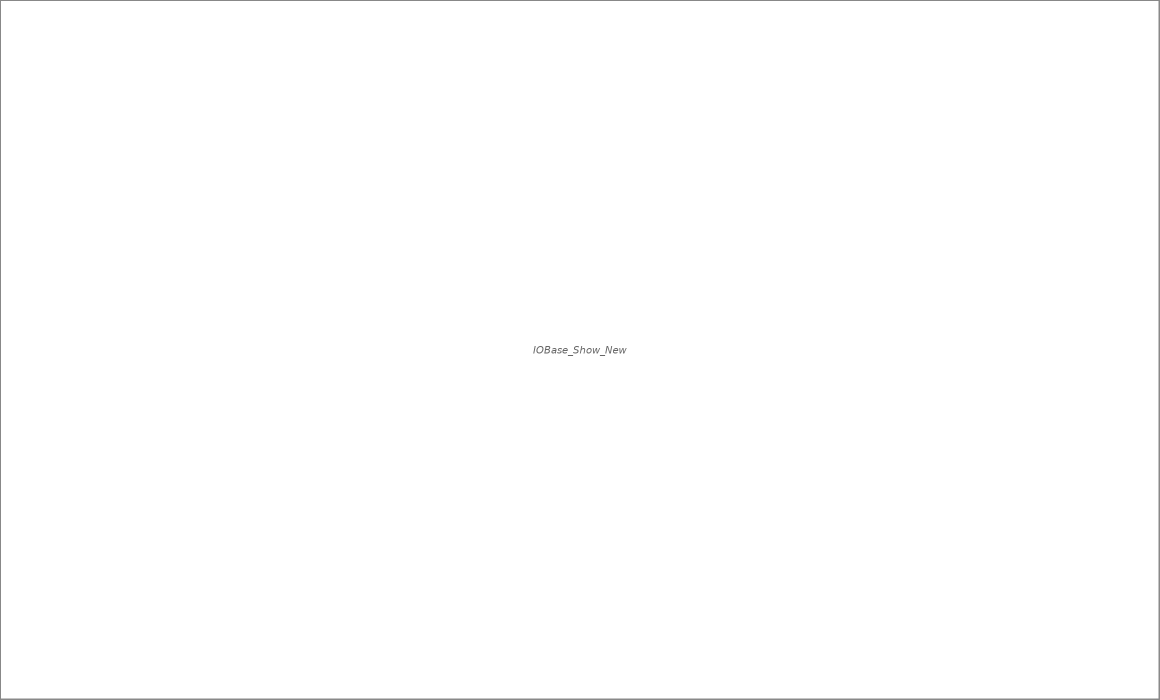
VISUALIZATION IO_Output  // 1160x700
    TabControl (0,0 1160x700)
        shows IOBase_Show_New(userData := TesterIO.fbIOBase_Output.HMIITF)
        [0]: TabTitle=Output
END_VISUALIZATION

// ---- VISUs/Loadding.TcVIS
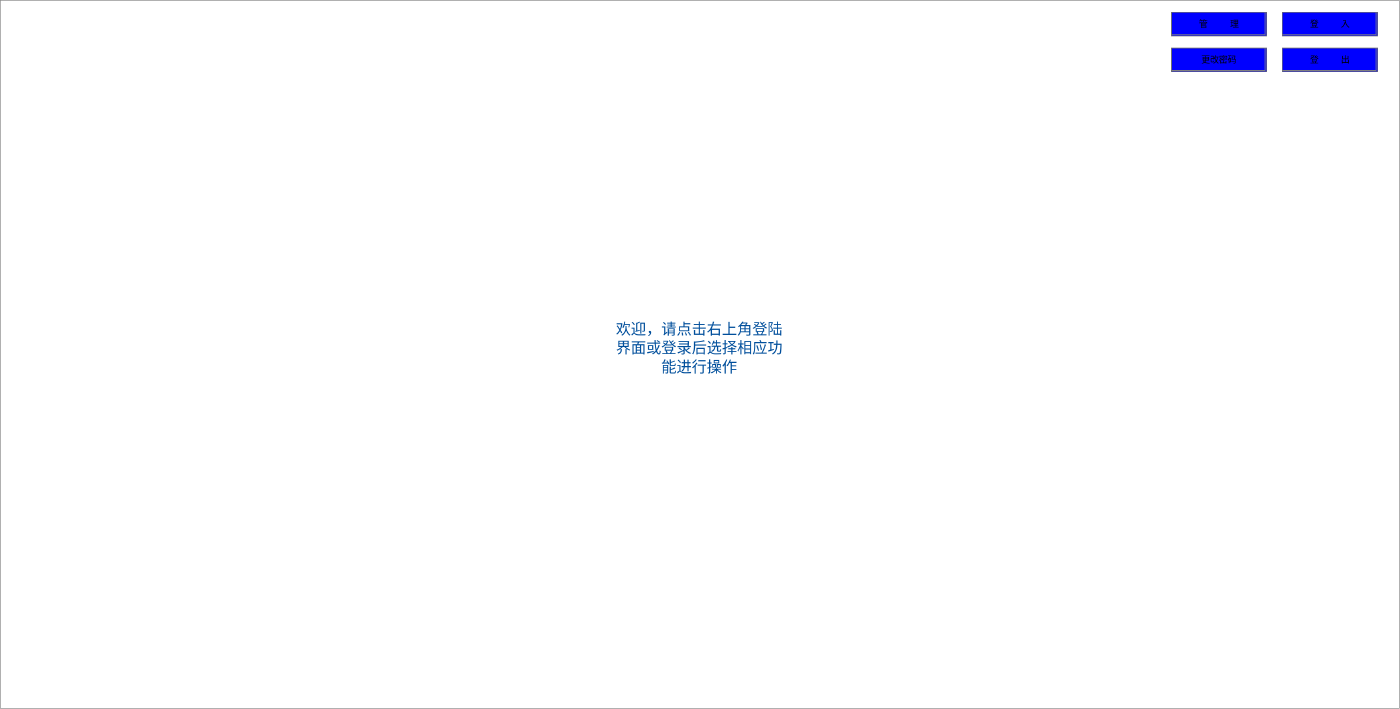
VISUALIZATION Loadding  // 1755x890, background image ImagePool1.Loadding
    Button (1607,15 120x30), "登 入"
        OnMouseClick: VisuUserMgmt Type=Login
        OnMouseClick: write the text variable via Default
    Button (1468,15 120x30), "管 理"
        OnMouseClick: VisuUserMgmt Type=OpenUserConfiguration
        OnMouseClick: write the text variable via Default
    Button (1468,60 120x30), "更改密码"
        OnMouseClick: VisuUserMgmt Type=ChangeUserPassword
        OnMouseClick: write the text variable via Default
    Button (1607,60 120x30), "登 出"
        OnMouseClick: VisuUserMgmt Type=Logout
        OnMouseClick: write the text variable via Default
        OnMouseClick: execute { VisuUserManagement.g_VisuLoginProviderManager.m_arrLoginProvider[0].stUserName:=""; }
    Rectangle (634,378 485x117), "欢迎，请点击右上角登陆 界面或登录后选择相应功 能进行操作"
END_VISUALIZATION

// ---- VISUs/Log/LogInf.TcVIS
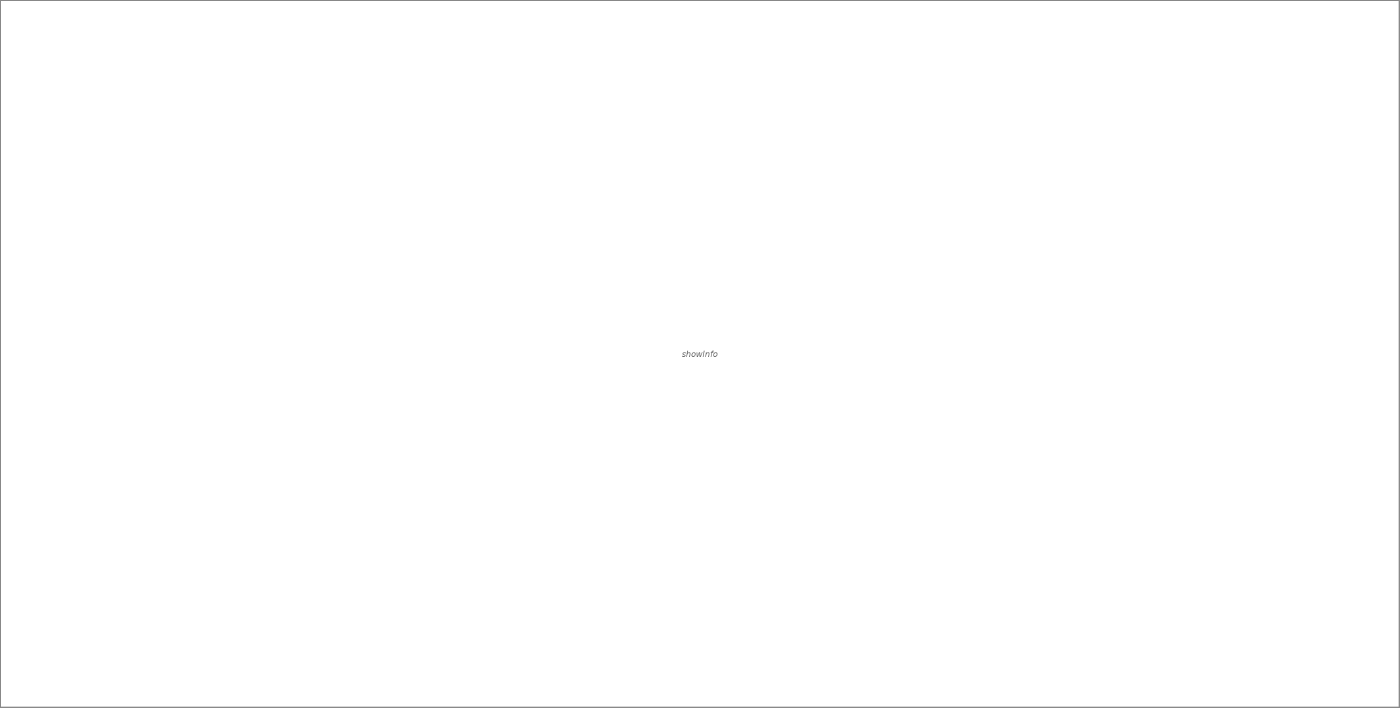
VISUALIZATION LogInf  // 1740x880
    TabControl (0,0 1740x880)
        shows showInfo(userData := gLog.HMIData)
        shows showInfo(userData := gDataChangeLog.HMIData)
        shows showInfo(userData := gDownTimeLog.HMIData)
        shows showInfo(userData := gBreakTimeLog.HMIData)
        shows showInfo(userData := gOperatorLog.HMIData)
        shows showInfo(userData := gRunningLog.HMIData)
        [1]: TabTitle=Data Change
        [2]: TabTitle=Error
        [3]: TabTitle=Time
        [4]: TabTitle=Operator
        [5]: TabTitle=Runing
END_VISUALIZATION

// ---- VISUs/Main.TcVIS
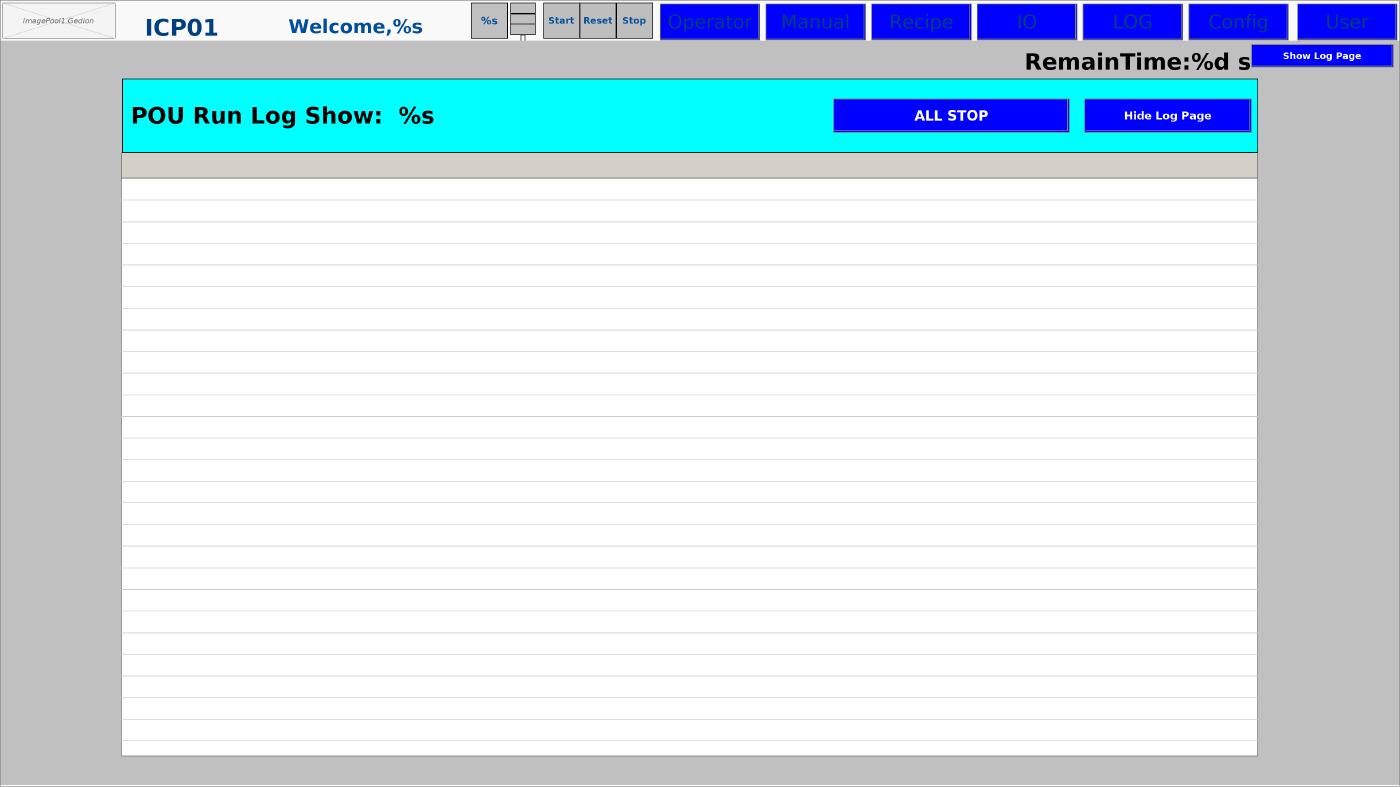
VISUALIZATION Main  // 1920x1080, background image ImagePool1.background
    Frame (0,0 1920x1077)
        shows MainFrame(userData := MainFramDUT)
    Frame (0,95 1920x984)
        shows Loadding()
        shows Manual()
        shows Config()
        shows IO()
        shows LogInf()
        shows Recipe()
        shows Operator()
    Button (1050,5 137x50), "Manual"
        OnMouseClick: execute {
            //MAIN.changePage(1);
        }
        OnMouseClick: FrameSelectionChange Selection=SelectedFrame=81912e38-ebf1-4b8c-bf44-e4a6c92ae24e, Selection=1, GlobSel=AssignType=Directly, SelType=Locally
    Button (1195,5 137x50), "Recipe"
        OnMouseClick: execute {
            //MAIN.changePage(1);
        }
        OnMouseClick: FrameSelectionChange Selection=SelectedFrame=81912e38-ebf1-4b8c-bf44-e4a6c92ae24e, Selection=5, GlobSel=AssignType=Directly, SelType=Locally
    Button (1485,5 137x50), "LOG"
        OnMouseClick: execute {
            //MAIN.changePage(1);
        }
        OnMouseClick: FrameSelectionChange Selection=SelectedFrame=81912e38-ebf1-4b8c-bf44-e4a6c92ae24e, Selection=4, GlobSel=AssignType=Directly, SelType=Locally
    Button (1630,5 137x50), "Config"
        OnMouseClick: execute {
            //MAIN.changePage(1);
        }
        OnMouseClick: FrameSelectionChange Selection=SelectedFrame=81912e38-ebf1-4b8c-bf44-e4a6c92ae24e, Selection=2, GlobSel=AssignType=Directly, SelType=Locally
    Button (1340,5 137x50), "IO"
        OnMouseClick: execute {
            //MAIN.changePage(1);
        }
        OnMouseClick: FrameSelectionChange Selection=SelectedFrame=81912e38-ebf1-4b8c-bf44-e4a6c92ae24e, Selection=3, GlobSel=AssignType=Directly, SelType=Locally
    Button (1779,5 137x50), "User"
        OnMouseClick: execute {
            //MAIN.changePage(1);
        }
        OnMouseClick: FrameSelectionChange Selection=SelectedFrame=81912e38-ebf1-4b8c-bf44-e4a6c92ae24e, GlobSel=AssignType=Directly, SelType=Locally
    Button (905,5 137x50), "Operator"
        OnMouseClick: execute {
            //MAIN.changePage(1);
        }
        OnMouseClick: FrameSelectionChange Selection=SelectedFrame=81912e38-ebf1-4b8c-bf44-e4a6c92ae24e, Selection=6, GlobSel=AssignType=Directly, SelType=Locally
    Frame (0,56 1920x1021), invisible if: (Not gSPOUBusy AND Not gShowPOURunLog) OR ( gSPOUBusy AND Not gShowPOURunLog)
        shows showInfo_Auto(userData := gRunningLog.HMIData)
    Button (1716,61 195x31), "Show Log Page", invisible if: gShowPOURunLog or Not gSPOUBusy
        OnMouseClick: execute { gShowPOURunLog:=NOT gShowPOURunLog; }
END_VISUALIZATION

// ---- VISUs/Operator/Operator.TcVIS
